ABB RAPID module: c1599a78.mod

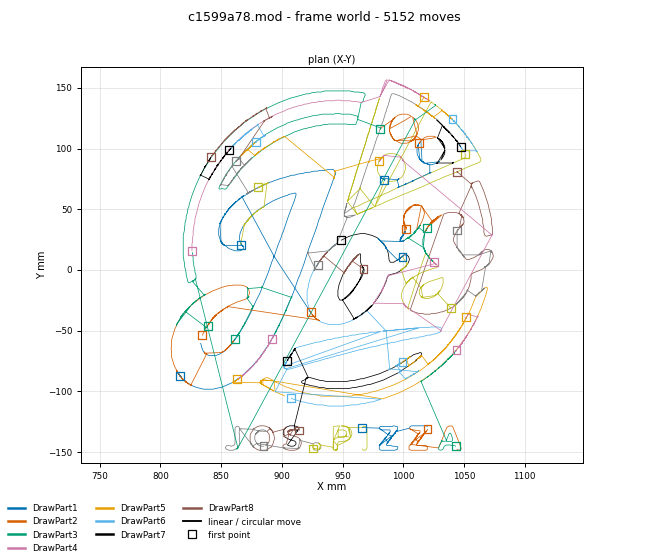
[picture p0: tool path of c1599a78.mod in frame world, 5152 of 5154 moves have a stored position in this frame; points joined in program order, loops and branches not executed]
MODULE ImageDraw
  ! Generated 2026-10-07 06:19 for ABB IRB 1600-10/1.45: 481 strokes
  ! Page 500 x 350 mm. Work object wPaper: Z points up, so pen-up is +Z and the tool uses orientation [0,1,0,0].
  PERS tooldata tPen:=[TRUE,[[0,0,120],[1,0,0,0]],[0.3,[0,0,60],[1,0,0,0],0,0,0]];
  PERS wobjdata wPaper:=[FALSE,TRUE,"",[[700,-175,0],[1,0,0,0]],[[0,0,0],[1,0,0,0]]];
  CONST robtarget pOrigin:=[[0,0,0],[0,1,0,0],[0,0,0,0],[9E9,9E9,9E9,9E9,9E9,9E9]];
  CONST jointtarget jHome:=[[0,0,0,0,30,0],[9E9,9E9,9E9,9E9,9E9,9E9]];
  CONST speeddata vTravel:=[250,200,5000,1000];

  PROC DrawImage()
    SingArea\Wrist;
    ConfL\Off;
    ConfJ\Off;
    MoveAbsJ jHome\NoEOffs,vTravel,fine,tPen;
    DrawPart1;
    DrawPart2;
    DrawPart3;
    DrawPart4;
    DrawPart5;
    DrawPart6;
    DrawPart7;
    DrawPart8;
    DrawPart9;
    DrawPart10;
    DrawPart11;
    DrawPart12;
    DrawPart13;
    DrawPart14;
    DrawPart15;
    DrawPart16;
    DrawPart17;
    DrawPart18;
    DrawPart19;
    DrawPart20;
    DrawPart21;
    DrawPart22;
    DrawPart23;
    DrawPart24;
    DrawPart25;
    DrawPart26;
    DrawPart27;
    DrawPart28;
    DrawPart29;
    DrawPart30;
    DrawPart31;
    DrawPart32;
    DrawPart33;
    DrawPart34;
    DrawPart35;
    DrawPart36;
    DrawPart37;
    DrawPart38;
    DrawPart39;
    DrawPart40;
    DrawPart41;
    DrawPart42;
    DrawPart43;
    MoveAbsJ jHome\NoEOffs,vTravel,fine,tPen;
  ENDPROC

  PROC DrawPart1()
    MoveL Offs(pOrigin,115.92,87.85,6.00),vTravel,z5,tPen\WObj:=wPaper;
    MoveL Offs(pOrigin,115.92,87.85,0.00),v60,z0,tPen\WObj:=wPaper;
    MoveL Offs(pOrigin,116.87,86.89,0.00),v40,z0,tPen\WObj:=wPaper;
    MoveL Offs(pOrigin,116.87,87.37,0.00),v40,z0,tPen\WObj:=wPaper;
    MoveL Offs(pOrigin,116.39,87.37,0.00),v40,z0,tPen\WObj:=wPaper;
    MoveL Offs(pOrigin,115.92,87.85,0.00),v40,z0,tPen\WObj:=wPaper;
    MoveL Offs(pOrigin,116.87,86.89,0.00),v40,z0,tPen\WObj:=wPaper;
    MoveL Offs(pOrigin,116.87,87.37,0.00),v40,z0,tPen\WObj:=wPaper;
    MoveL Offs(pOrigin,116.39,87.37,0.00),v40,z0,tPen\WObj:=wPaper;
    MoveL Offs(pOrigin,115.92,87.85,0.00),v40,z0,tPen\WObj:=wPaper;
    MoveL Offs(pOrigin,115.44,88.80,0.00),v40,z0,tPen\WObj:=wPaper;
    MoveL Offs(pOrigin,115.44,89.28,0.00),v40,z0,tPen\WObj:=wPaper;
    MoveL Offs(pOrigin,114.96,89.28,0.00),v40,z0,tPen\WObj:=wPaper;
    MoveL Offs(pOrigin,114.48,89.76,0.00),v40,z0,tPen\WObj:=wPaper;
    MoveL Offs(pOrigin,115.44,88.80,0.00),v40,z0,tPen\WObj:=wPaper;
    MoveL Offs(pOrigin,115.44,89.28,0.00),v40,z0,tPen\WObj:=wPaper;
    MoveL Offs(pOrigin,114.96,89.28,0.00),v40,z0,tPen\WObj:=wPaper;
    MoveL Offs(pOrigin,114.48,89.76,0.00),v40,z0,tPen\WObj:=wPaper;
    MoveL Offs(pOrigin,115.44,88.80,0.00),v40,fine,tPen\WObj:=wPaper;
    MoveL Offs(pOrigin,115.44,88.80,6.00),v60,z5,tPen\WObj:=wPaper;
    MoveL Offs(pOrigin,114.32,90.72,6.00),vTravel,z5,tPen\WObj:=wPaper;
    MoveL Offs(pOrigin,114.32,90.72,0.00),v60,z0,tPen\WObj:=wPaper;
    MoveL Offs(pOrigin,117.83,85.93,0.00),v40,z0,tPen\WObj:=wPaper;
    MoveL Offs(pOrigin,121.66,82.58,0.00),v40,z0,tPen\WObj:=wPaper;
    MoveL Offs(pOrigin,126.45,79.54,0.00),v40,z0,tPen\WObj:=wPaper;
    MoveL Offs(pOrigin,129.80,78.27,0.00),v40,z0,tPen\WObj:=wPaper;
    MoveL Offs(pOrigin,135.55,76.83,0.00),v40,z0,tPen\WObj:=wPaper;
    MoveL Offs(pOrigin,143.21,76.83,0.00),v40,z0,tPen\WObj:=wPaper;
    MoveL Offs(pOrigin,150.87,78.59,0.00),v40,z0,tPen\WObj:=wPaper;
    MoveL Offs(pOrigin,158.54,81.94,0.00),v40,z0,tPen\WObj:=wPaper;
    MoveL Offs(pOrigin,166.68,87.37,0.00),v40,z0,tPen\WObj:=wPaper;
    MoveL Offs(pOrigin,176.25,96.46,0.00),v40,z0,tPen\WObj:=wPaper;
    MoveL Offs(pOrigin,181.52,102.69,0.00),v40,z0,tPen\WObj:=wPaper;
    MoveL Offs(pOrigin,189.50,114.18,0.00),v40,z0,tPen\WObj:=wPaper;
    MoveL Offs(pOrigin,194.13,122.80,0.00),v40,z0,tPen\WObj:=wPaper;
    MoveL Offs(pOrigin,200.36,135.25,0.00),v40,z0,tPen\WObj:=wPaper;
    MoveL Offs(pOrigin,209.46,156.32,0.00),v40,z0,tPen\WObj:=wPaper;
    MoveL Offs(pOrigin,213.77,168.77,0.00),v40,z0,tPen\WObj:=wPaper;
    MoveL Offs(pOrigin,214.40,169.73,0.00),v40,z0,tPen\WObj:=wPaper;
    MoveL Offs(pOrigin,218.08,179.79,0.00),v40,z0,tPen\WObj:=wPaper;
    MoveL Offs(pOrigin,222.07,192.24,0.00),v40,z0,tPen\WObj:=wPaper;
    MoveL Offs(pOrigin,228.61,209.96,0.00),v40,z0,tPen\WObj:=wPaper;
    MoveL Offs(pOrigin,230.37,216.18,0.00),v40,z0,tPen\WObj:=wPaper;
    MoveL Offs(pOrigin,231.16,217.62,0.00),v40,z0,tPen\WObj:=wPaper;
    MoveL Offs(pOrigin,234.04,226.72,0.00),v40,z0,tPen\WObj:=wPaper;
    MoveL Offs(pOrigin,242.02,248.27,0.00),v40,z0,tPen\WObj:=wPaper;
    MoveL Offs(pOrigin,242.66,250.66,0.00),v40,z0,tPen\WObj:=wPaper;
    MoveL Offs(pOrigin,244.25,254.01,0.00),v40,z0,tPen\WObj:=wPaper;
    MoveL Offs(pOrigin,244.09,255.93,0.00),v40,z0,tPen\WObj:=wPaper;
    MoveL Offs(pOrigin,242.34,257.69,0.00),v40,z0,tPen\WObj:=wPaper;
    MoveL Offs(pOrigin,238.51,257.85,0.00),v40,z0,tPen\WObj:=wPaper;
    MoveL Offs(pOrigin,234.68,256.89,0.00),v40,z0,tPen\WObj:=wPaper;
    MoveL Offs(pOrigin,230.85,256.89,0.00),v40,z0,tPen\WObj:=wPaper;
    MoveL Offs(pOrigin,229.41,256.41,0.00),v40,z0,tPen\WObj:=wPaper;
    MoveL Offs(pOrigin,226.54,256.41,0.00),v40,z0,tPen\WObj:=wPaper;
    MoveL Offs(pOrigin,222.70,255.45,0.00),v40,z0,tPen\WObj:=wPaper;
    MoveL Offs(pOrigin,220.31,255.45,0.00),v40,z0,tPen\WObj:=wPaper;
    MoveL Offs(pOrigin,216.96,254.49,0.00),v40,z0,tPen\WObj:=wPaper;
    MoveL Offs(pOrigin,213.13,254.01,0.00),v40,z0,tPen\WObj:=wPaper;
    MoveL Offs(pOrigin,210.25,253.06,0.00),v40,z0,tPen\WObj:=wPaper;
    MoveL Offs(pOrigin,208.34,253.06,0.00),v40,z0,tPen\WObj:=wPaper;
    MoveL Offs(pOrigin,200.68,250.66,0.00),v40,z0,tPen\WObj:=wPaper;
    MoveL Offs(pOrigin,199.72,250.66,0.00),v40,z0,tPen\WObj:=wPaper;
    MoveL Offs(pOrigin,189.66,246.99,0.00),v40,z0,tPen\WObj:=wPaper;
    MoveL Offs(pOrigin,181.04,242.84,0.00),v40,z0,tPen\WObj:=wPaper;
    MoveL Offs(pOrigin,179.13,242.20,0.00),v40,z0,tPen\WObj:=wPaper;
    MoveL Offs(pOrigin,167.15,234.86,0.00),v40,z0,tPen\WObj:=wPaper;
    MoveL Offs(pOrigin,162.37,231.03,0.00),v40,z0,tPen\WObj:=wPaper;
    MoveL Offs(pOrigin,156.62,225.28,0.00),v40,z0,tPen\WObj:=wPaper;
    MoveL Offs(pOrigin,153.75,221.45,0.00),v40,z0,tPen\WObj:=wPaper;
    MoveL Offs(pOrigin,151.03,217.14,0.00),v40,z0,tPen\WObj:=wPaper;
    MoveL Offs(pOrigin,148.48,210.92,0.00),v40,z0,tPen\WObj:=wPaper;
    MoveL Offs(pOrigin,148.00,208.52,0.00),v40,z0,tPen\WObj:=wPaper;
    MoveL Offs(pOrigin,148.00,203.73,0.00),v40,z0,tPen\WObj:=wPaper;
    MoveL Offs(pOrigin,149.28,199.90,0.00),v40,z0,tPen\WObj:=wPaper;
    MoveL Offs(pOrigin,151.83,196.23,0.00),v40,z0,tPen\WObj:=wPaper;
    MoveL Offs(pOrigin,156.62,192.56,0.00),v40,z0,tPen\WObj:=wPaper;
    MoveL Offs(pOrigin,161.41,190.80,0.00),v40,z0,tPen\WObj:=wPaper;
    MoveL Offs(pOrigin,165.72,190.80,0.00),v40,z0,tPen\WObj:=wPaper;
    MoveL Offs(pOrigin,167.63,191.76,0.00),v40,z0,tPen\WObj:=wPaper;
    MoveL Offs(pOrigin,168.59,193.20,0.00),v40,z0,tPen\WObj:=wPaper;
    MoveL Offs(pOrigin,168.43,194.15,0.00),v40,z0,tPen\WObj:=wPaper;
    MoveL Offs(pOrigin,167.00,195.59,0.00),v40,z0,tPen\WObj:=wPaper;
    MoveL Offs(pOrigin,165.24,199.90,0.00),v40,z0,tPen\WObj:=wPaper;
    MoveL Offs(pOrigin,165.24,203.25,0.00),v40,z0,tPen\WObj:=wPaper;
    MoveL Offs(pOrigin,165.72,205.65,0.00),v40,z0,tPen\WObj:=wPaper;
    MoveL Offs(pOrigin,168.27,211.39,0.00),v40,z0,tPen\WObj:=wPaper;
    MoveL Offs(pOrigin,172.90,217.62,0.00),v40,z0,tPen\WObj:=wPaper;
    MoveL Offs(pOrigin,179.61,223.85,0.00),v40,z0,tPen\WObj:=wPaper;
    MoveL Offs(pOrigin,187.27,228.79,0.00),v40,z0,tPen\WObj:=wPaper;
    MoveL Offs(pOrigin,193.49,232.31,0.00),v40,z0,tPen\WObj:=wPaper;
    MoveL Offs(pOrigin,201.15,235.50,0.00),v40,z0,tPen\WObj:=wPaper;
    MoveL Offs(pOrigin,204.51,236.46,0.00),v40,z0,tPen\WObj:=wPaper;
    MoveL Offs(pOrigin,205.94,237.25,0.00),v40,z0,tPen\WObj:=wPaper;
    MoveL Offs(pOrigin,210.73,238.37,0.00),v40,z0,tPen\WObj:=wPaper;
    MoveL Offs(pOrigin,211.53,238.21,0.00),v40,z0,tPen\WObj:=wPaper;
    MoveL Offs(pOrigin,211.69,236.77,0.00),v40,z0,tPen\WObj:=wPaper;
    MoveL Offs(pOrigin,210.41,232.46,0.00),v40,z0,tPen\WObj:=wPaper;
    MoveL Offs(pOrigin,205.31,219.06,0.00),v40,z0,tPen\WObj:=wPaper;
    MoveL Offs(pOrigin,201.00,206.13,0.00),v40,z0,tPen\WObj:=wPaper;
    MoveL Offs(pOrigin,200.36,205.17,0.00),v40,z0,tPen\WObj:=wPaper;
    MoveL Offs(pOrigin,199.40,201.82,0.00),v40,z0,tPen\WObj:=wPaper;
    MoveL Offs(pOrigin,196.69,195.11,0.00),v40,z0,tPen\WObj:=wPaper;
    MoveL Offs(pOrigin,193.65,186.01,0.00),v40,z0,tPen\WObj:=wPaper;
    MoveL Offs(pOrigin,191.74,181.70,0.00),v40,z0,tPen\WObj:=wPaper;
    MoveL Offs(pOrigin,188.86,173.08,0.00),v40,z0,tPen\WObj:=wPaper;
    MoveL Offs(pOrigin,181.68,155.37,0.00),v40,z0,tPen\WObj:=wPaper;
    MoveL Offs(pOrigin,178.49,149.14,0.00),v40,z0,tPen\WObj:=wPaper;
    MoveL Offs(pOrigin,174.50,140.04,0.00),v40,z0,tPen\WObj:=wPaper;
    MoveL Offs(pOrigin,169.23,129.99,0.00),v40,z0,tPen\WObj:=wPaper;
    MoveL Offs(pOrigin,163.48,120.41,0.00),v40,z0,tPen\WObj:=wPaper;
    MoveL Offs(pOrigin,158.54,113.70,0.00),v40,z0,tPen\WObj:=wPaper;
    MoveL Offs(pOrigin,153.27,108.44,0.00),v40,z0,tPen\WObj:=wPaper;
    MoveL Offs(pOrigin,148.00,105.40,0.00),v40,z0,tPen\WObj:=wPaper;
    MoveL Offs(pOrigin,145.61,104.61,0.00),v40,z0,tPen\WObj:=wPaper;
    MoveL Offs(pOrigin,139.86,104.61,0.00),v40,z0,tPen\WObj:=wPaper;
    MoveL Offs(pOrigin,137.46,105.72,0.00),v40,z0,tPen\WObj:=wPaper;
    MoveL Offs(pOrigin,135.71,107.48,0.00),v40,z0,tPen\WObj:=wPaper;
    MoveL Offs(pOrigin,134.59,109.39,0.00),v40,z0,tPen\WObj:=wPaper;
    MoveL Offs(pOrigin,133.15,114.66,0.00),v40,z0,tPen\WObj:=wPaper;
  ENDPROC

  PROC DrawPart2()
    MoveL Offs(pOrigin,134.59,121.37,0.00),v40,z0,tPen\WObj:=wPaper;
    MoveL Offs(pOrigin,137.15,127.11,0.00),v40,z0,tPen\WObj:=wPaper;
    MoveL Offs(pOrigin,143.21,135.73,0.00),v40,z0,tPen\WObj:=wPaper;
    MoveL Offs(pOrigin,145.61,138.13,0.00),v40,z0,tPen\WObj:=wPaper;
    MoveL Offs(pOrigin,149.92,141.48,0.00),v40,z0,tPen\WObj:=wPaper;
    MoveL Offs(pOrigin,155.66,145.15,0.00),v40,z0,tPen\WObj:=wPaper;
    MoveL Offs(pOrigin,162.85,148.50,0.00),v40,z0,tPen\WObj:=wPaper;
    MoveL Offs(pOrigin,170.03,150.90,0.00),v40,z0,tPen\WObj:=wPaper;
    MoveL Offs(pOrigin,172.42,152.97,0.00),v40,z0,tPen\WObj:=wPaper;
    MoveL Offs(pOrigin,173.38,156.32,0.00),v40,z0,tPen\WObj:=wPaper;
    MoveL Offs(pOrigin,172.58,159.20,0.00),v40,z0,tPen\WObj:=wPaper;
    MoveL Offs(pOrigin,170.51,161.43,0.00),v40,z0,tPen\WObj:=wPaper;
    MoveL Offs(pOrigin,166.68,162.55,0.00),v40,z0,tPen\WObj:=wPaper;
    MoveL Offs(pOrigin,159.97,162.55,0.00),v40,z0,tPen\WObj:=wPaper;
    MoveL Offs(pOrigin,158.54,162.07,0.00),v40,z0,tPen\WObj:=wPaper;
    MoveL Offs(pOrigin,155.66,162.07,0.00),v40,z0,tPen\WObj:=wPaper;
    MoveL Offs(pOrigin,150.87,160.79,0.00),v40,z0,tPen\WObj:=wPaper;
    MoveL Offs(pOrigin,142.25,157.44,0.00),v40,z0,tPen\WObj:=wPaper;
    MoveL Offs(pOrigin,135.07,153.45,0.00),v40,z0,tPen\WObj:=wPaper;
    MoveL Offs(pOrigin,125.01,145.79,0.00),v40,z0,tPen\WObj:=wPaper;
    MoveL Offs(pOrigin,124.06,144.35,0.00),v40,z0,tPen\WObj:=wPaper;
    MoveL Offs(pOrigin,118.79,138.61,0.00),v40,z0,tPen\WObj:=wPaper;
    MoveL Offs(pOrigin,115.28,133.34,0.00),v40,z0,tPen\WObj:=wPaper;
    MoveL Offs(pOrigin,111.77,126.15,0.00),v40,z0,tPen\WObj:=wPaper;
    MoveL Offs(pOrigin,109.21,117.54,0.00),v40,z0,tPen\WObj:=wPaper;
    MoveL Offs(pOrigin,109.21,111.79,0.00),v40,z0,tPen\WObj:=wPaper;
    MoveL Offs(pOrigin,108.73,110.35,0.00),v40,z0,tPen\WObj:=wPaper;
    MoveL Offs(pOrigin,109.21,108.44,0.00),v40,z0,tPen\WObj:=wPaper;
    MoveL Offs(pOrigin,109.21,103.17,0.00),v40,z0,tPen\WObj:=wPaper;
    MoveL Offs(pOrigin,111.45,95.99,0.00),v40,z0,tPen\WObj:=wPaper;
    MoveL Offs(pOrigin,114.32,90.72,0.00),v40,fine,tPen\WObj:=wPaper;
    MoveL Offs(pOrigin,114.32,90.72,6.00),v60,z5,tPen\WObj:=wPaper;
    MoveL Offs(pOrigin,113.52,91.68,6.00),vTravel,z5,tPen\WObj:=wPaper;
    MoveL Offs(pOrigin,113.52,91.68,0.00),v60,z0,tPen\WObj:=wPaper;
    MoveL Offs(pOrigin,113.52,92.15,0.00),v40,z0,tPen\WObj:=wPaper;
    MoveL Offs(pOrigin,113.04,92.15,0.00),v40,z0,tPen\WObj:=wPaper;
    MoveL Offs(pOrigin,113.52,91.68,0.00),v40,z0,tPen\WObj:=wPaper;
    MoveL Offs(pOrigin,113.52,92.15,0.00),v40,z0,tPen\WObj:=wPaper;
    MoveL Offs(pOrigin,113.04,92.15,0.00),v40,z0,tPen\WObj:=wPaper;
    MoveL Offs(pOrigin,113.52,91.68,0.00),v40,fine,tPen\WObj:=wPaper;
    MoveL Offs(pOrigin,113.52,91.68,6.00),v60,z5,tPen\WObj:=wPaper;
    MoveL Offs(pOrigin,117.35,85.93,6.00),vTravel,z5,tPen\WObj:=wPaper;
    MoveL Offs(pOrigin,117.35,85.93,0.00),v60,z0,tPen\WObj:=wPaper;
    MoveL Offs(pOrigin,119.27,84.01,0.00),v40,z0,tPen\WObj:=wPaper;
    MoveL Offs(pOrigin,119.27,84.49,0.00),v40,z0,tPen\WObj:=wPaper;
    MoveL Offs(pOrigin,118.79,84.49,0.00),v40,z0,tPen\WObj:=wPaper;
    MoveL Offs(pOrigin,117.35,85.93,0.00),v40,z0,tPen\WObj:=wPaper;
    MoveL Offs(pOrigin,119.27,84.01,0.00),v40,z0,tPen\WObj:=wPaper;
    MoveL Offs(pOrigin,119.27,84.49,0.00),v40,z0,tPen\WObj:=wPaper;
    MoveL Offs(pOrigin,118.79,84.49,0.00),v40,z0,tPen\WObj:=wPaper;
    MoveL Offs(pOrigin,117.35,85.93,0.00),v40,fine,tPen\WObj:=wPaper;
    MoveL Offs(pOrigin,117.35,85.93,6.00),v60,z5,tPen\WObj:=wPaper;
    MoveL Offs(pOrigin,120.23,83.54,6.00),vTravel,z5,tPen\WObj:=wPaper;
    MoveL Offs(pOrigin,120.23,83.54,0.00),v60,z0,tPen\WObj:=wPaper;
    MoveL Offs(pOrigin,121.66,82.10,0.00),v40,z0,tPen\WObj:=wPaper;
    MoveL Offs(pOrigin,121.66,82.58,0.00),v40,z0,tPen\WObj:=wPaper;
    MoveL Offs(pOrigin,121.18,82.58,0.00),v40,z0,tPen\WObj:=wPaper;
    MoveL Offs(pOrigin,120.23,83.54,0.00),v40,z0,tPen\WObj:=wPaper;
    MoveL Offs(pOrigin,121.66,82.10,0.00),v40,z0,tPen\WObj:=wPaper;
    MoveL Offs(pOrigin,121.66,82.58,0.00),v40,z0,tPen\WObj:=wPaper;
    MoveL Offs(pOrigin,121.18,82.58,0.00),v40,z0,tPen\WObj:=wPaper;
    MoveL Offs(pOrigin,120.23,83.54,0.00),v40,fine,tPen\WObj:=wPaper;
    MoveL Offs(pOrigin,120.23,83.54,6.00),v60,z5,tPen\WObj:=wPaper;
    MoveL Offs(pOrigin,122.62,81.62,6.00),vTravel,z5,tPen\WObj:=wPaper;
    MoveL Offs(pOrigin,122.62,81.62,0.00),v60,z0,tPen\WObj:=wPaper;
    MoveL Offs(pOrigin,123.10,81.14,0.00),v40,z0,tPen\WObj:=wPaper;
    MoveL Offs(pOrigin,123.10,81.62,0.00),v40,z0,tPen\WObj:=wPaper;
    MoveL Offs(pOrigin,122.62,81.62,0.00),v40,z0,tPen\WObj:=wPaper;
    MoveL Offs(pOrigin,123.10,81.14,0.00),v40,z0,tPen\WObj:=wPaper;
    MoveL Offs(pOrigin,123.10,81.62,0.00),v40,z0,tPen\WObj:=wPaper;
    MoveL Offs(pOrigin,122.62,81.62,0.00),v40,fine,tPen\WObj:=wPaper;
    MoveL Offs(pOrigin,122.62,81.62,6.00),v60,z5,tPen\WObj:=wPaper;
    MoveL Offs(pOrigin,125.01,80.18,6.00),vTravel,z5,tPen\WObj:=wPaper;
    MoveL Offs(pOrigin,125.01,80.18,0.00),v60,z0,tPen\WObj:=wPaper;
    MoveL Offs(pOrigin,125.49,79.70,0.00),v40,z0,tPen\WObj:=wPaper;
    MoveL Offs(pOrigin,125.49,80.18,0.00),v40,z0,tPen\WObj:=wPaper;
    MoveL Offs(pOrigin,125.01,80.18,0.00),v40,z0,tPen\WObj:=wPaper;
    MoveL Offs(pOrigin,125.49,79.70,0.00),v40,z0,tPen\WObj:=wPaper;
    MoveL Offs(pOrigin,125.49,80.18,0.00),v40,z0,tPen\WObj:=wPaper;
    MoveL Offs(pOrigin,125.01,80.18,0.00),v40,fine,tPen\WObj:=wPaper;
    MoveL Offs(pOrigin,125.01,80.18,6.00),v60,z5,tPen\WObj:=wPaper;
    MoveL Offs(pOrigin,137.94,105.56,6.00),vTravel,z5,tPen\WObj:=wPaper;
    MoveL Offs(pOrigin,137.94,105.56,0.00),v60,z0,tPen\WObj:=wPaper;
    MoveL Offs(pOrigin,138.42,105.56,0.00),v40,z0,tPen\WObj:=wPaper;
    MoveL Offs(pOrigin,137.46,106.04,0.00),v40,z0,tPen\WObj:=wPaper;
    MoveL Offs(pOrigin,137.94,105.56,0.00),v40,z0,tPen\WObj:=wPaper;
    MoveL Offs(pOrigin,138.42,105.56,0.00),v40,z0,tPen\WObj:=wPaper;
    MoveL Offs(pOrigin,137.46,106.04,0.00),v40,z0,tPen\WObj:=wPaper;
    MoveL Offs(pOrigin,137.94,105.56,0.00),v40,fine,tPen\WObj:=wPaper;
    MoveL Offs(pOrigin,137.94,105.56,6.00),v60,z5,tPen\WObj:=wPaper;
    MoveL Offs(pOrigin,136.51,106.52,6.00),vTravel,z5,tPen\WObj:=wPaper;
    MoveL Offs(pOrigin,136.51,106.52,0.00),v60,z0,tPen\WObj:=wPaper;
    MoveL Offs(pOrigin,136.03,107.48,0.00),v40,z0,tPen\WObj:=wPaper;
    MoveL Offs(pOrigin,136.51,107.00,0.00),v40,z0,tPen\WObj:=wPaper;
    MoveL Offs(pOrigin,136.51,106.52,0.00),v40,z0,tPen\WObj:=wPaper;
    MoveL Offs(pOrigin,136.03,107.48,0.00),v40,z0,tPen\WObj:=wPaper;
    MoveL Offs(pOrigin,136.51,107.00,0.00),v40,z0,tPen\WObj:=wPaper;
    MoveL Offs(pOrigin,136.51,106.52,0.00),v40,fine,tPen\WObj:=wPaper;
    MoveL Offs(pOrigin,136.51,106.52,6.00),v60,z5,tPen\WObj:=wPaper;
    MoveL Offs(pOrigin,150.39,107.00,6.00),vTravel,z5,tPen\WObj:=wPaper;
    MoveL Offs(pOrigin,150.39,107.00,0.00),v60,z0,tPen\WObj:=wPaper;
    MoveL Offs(pOrigin,150.87,107.00,0.00),v40,z0,tPen\WObj:=wPaper;
    MoveL Offs(pOrigin,151.83,107.96,0.00),v40,z0,tPen\WObj:=wPaper;
    MoveL Offs(pOrigin,150.39,107.00,0.00),v40,z0,tPen\WObj:=wPaper;
    MoveL Offs(pOrigin,150.87,107.00,0.00),v40,z0,tPen\WObj:=wPaper;
    MoveL Offs(pOrigin,151.83,107.96,0.00),v40,z0,tPen\WObj:=wPaper;
    MoveL Offs(pOrigin,150.39,107.00,0.00),v40,fine,tPen\WObj:=wPaper;
    MoveL Offs(pOrigin,150.39,107.00,6.00),v60,z5,tPen\WObj:=wPaper;
    MoveL Offs(pOrigin,153.27,108.92,6.00),vTravel,z5,tPen\WObj:=wPaper;
    MoveL Offs(pOrigin,153.27,108.92,0.00),v60,z0,tPen\WObj:=wPaper;
    MoveL Offs(pOrigin,157.58,113.23,0.00),v40,z0,tPen\WObj:=wPaper;
    MoveL Offs(pOrigin,153.27,108.92,0.00),v40,fine,tPen\WObj:=wPaper;
    MoveL Offs(pOrigin,153.27,108.92,6.00),v60,z5,tPen\WObj:=wPaper;
    MoveL Offs(pOrigin,158.54,114.18,6.00),vTravel,z5,tPen\WObj:=wPaper;
    MoveL Offs(pOrigin,158.54,114.18,0.00),v60,z0,tPen\WObj:=wPaper;
    MoveL Offs(pOrigin,159.97,116.10,0.00),v40,z0,tPen\WObj:=wPaper;
    MoveL Offs(pOrigin,158.54,114.18,0.00),v40,fine,tPen\WObj:=wPaper;
    MoveL Offs(pOrigin,158.54,114.18,6.00),v60,z5,tPen\WObj:=wPaper;
    MoveL Offs(pOrigin,160.45,117.06,6.00),vTravel,z5,tPen\WObj:=wPaper;
    MoveL Offs(pOrigin,160.45,117.06,0.00),v60,z0,tPen\WObj:=wPaper;
  ENDPROC

  PROC DrawPart3()
    MoveL Offs(pOrigin,161.41,118.01,0.00),v40,z0,tPen\WObj:=wPaper;
    MoveL Offs(pOrigin,160.45,117.06,0.00),v40,fine,tPen\WObj:=wPaper;
    MoveL Offs(pOrigin,160.45,117.06,6.00),v60,z5,tPen\WObj:=wPaper;
    MoveL Offs(pOrigin,163.32,120.89,6.00),vTravel,z5,tPen\WObj:=wPaper;
    MoveL Offs(pOrigin,163.32,120.89,0.00),v60,z0,tPen\WObj:=wPaper;
    MoveL Offs(pOrigin,163.80,121.37,0.00),v40,z0,tPen\WObj:=wPaper;
    MoveL Offs(pOrigin,163.80,121.85,0.00),v40,z0,tPen\WObj:=wPaper;
    MoveL Offs(pOrigin,163.32,120.89,0.00),v40,z0,tPen\WObj:=wPaper;
    MoveL Offs(pOrigin,163.80,121.37,0.00),v40,z0,tPen\WObj:=wPaper;
    MoveL Offs(pOrigin,163.80,121.85,0.00),v40,z0,tPen\WObj:=wPaper;
    MoveL Offs(pOrigin,163.32,120.89,0.00),v40,fine,tPen\WObj:=wPaper;
    MoveL Offs(pOrigin,163.32,120.89,6.00),v60,z5,tPen\WObj:=wPaper;
    MoveL Offs(pOrigin,164.28,122.32,6.00),vTravel,z5,tPen\WObj:=wPaper;
    MoveL Offs(pOrigin,164.28,122.32,0.00),v60,z0,tPen\WObj:=wPaper;
    MoveL Offs(pOrigin,164.76,122.80,0.00),v40,z0,tPen\WObj:=wPaper;
    MoveL Offs(pOrigin,164.76,123.28,0.00),v40,z0,tPen\WObj:=wPaper;
    MoveL Offs(pOrigin,164.28,122.32,0.00),v40,z0,tPen\WObj:=wPaper;
    MoveL Offs(pOrigin,164.76,122.80,0.00),v40,z0,tPen\WObj:=wPaper;
    MoveL Offs(pOrigin,164.76,123.28,0.00),v40,z0,tPen\WObj:=wPaper;
    MoveL Offs(pOrigin,164.28,122.32,0.00),v40,fine,tPen\WObj:=wPaper;
    MoveL Offs(pOrigin,164.28,122.32,6.00),v60,z5,tPen\WObj:=wPaper;
    MoveL Offs(pOrigin,167.63,128.07,6.00),vTravel,z5,tPen\WObj:=wPaper;
    MoveL Offs(pOrigin,167.63,128.07,0.00),v60,z0,tPen\WObj:=wPaper;
    MoveL Offs(pOrigin,168.59,129.51,0.00),v40,z0,tPen\WObj:=wPaper;
    MoveL Offs(pOrigin,167.63,128.07,0.00),v40,fine,tPen\WObj:=wPaper;
    MoveL Offs(pOrigin,167.63,128.07,6.00),v60,z5,tPen\WObj:=wPaper;
    MoveL Offs(pOrigin,169.07,130.46,6.00),vTravel,z5,tPen\WObj:=wPaper;
    MoveL Offs(pOrigin,169.07,130.46,0.00),v60,z0,tPen\WObj:=wPaper;
    MoveL Offs(pOrigin,169.55,130.94,0.00),v40,z0,tPen\WObj:=wPaper;
    MoveL Offs(pOrigin,169.55,131.42,0.00),v40,z0,tPen\WObj:=wPaper;
    MoveL Offs(pOrigin,169.07,130.46,0.00),v40,z0,tPen\WObj:=wPaper;
    MoveL Offs(pOrigin,169.55,130.94,0.00),v40,z0,tPen\WObj:=wPaper;
    MoveL Offs(pOrigin,169.55,131.42,0.00),v40,z0,tPen\WObj:=wPaper;
    MoveL Offs(pOrigin,169.07,130.46,0.00),v40,fine,tPen\WObj:=wPaper;
    MoveL Offs(pOrigin,169.07,130.46,6.00),v60,z5,tPen\WObj:=wPaper;
    MoveL Offs(pOrigin,175.30,142.92,6.00),vTravel,z5,tPen\WObj:=wPaper;
    MoveL Offs(pOrigin,175.30,142.92,0.00),v60,z0,tPen\WObj:=wPaper;
    MoveL Offs(pOrigin,175.77,143.39,0.00),v40,z0,tPen\WObj:=wPaper;
    MoveL Offs(pOrigin,175.77,143.87,0.00),v40,z0,tPen\WObj:=wPaper;
    MoveL Offs(pOrigin,175.30,142.92,0.00),v40,z0,tPen\WObj:=wPaper;
    MoveL Offs(pOrigin,175.77,143.39,0.00),v40,z0,tPen\WObj:=wPaper;
    MoveL Offs(pOrigin,175.77,143.87,0.00),v40,z0,tPen\WObj:=wPaper;
    MoveL Offs(pOrigin,175.30,142.92,0.00),v40,fine,tPen\WObj:=wPaper;
    MoveL Offs(pOrigin,175.30,142.92,6.00),v60,z5,tPen\WObj:=wPaper;
    MoveL Offs(pOrigin,176.25,144.83,6.00),vTravel,z5,tPen\WObj:=wPaper;
    MoveL Offs(pOrigin,176.25,144.83,0.00),v60,z0,tPen\WObj:=wPaper;
    MoveL Offs(pOrigin,176.73,145.31,0.00),v40,z0,tPen\WObj:=wPaper;
    MoveL Offs(pOrigin,176.73,145.79,0.00),v40,z0,tPen\WObj:=wPaper;
    MoveL Offs(pOrigin,176.25,144.83,0.00),v40,z0,tPen\WObj:=wPaper;
    MoveL Offs(pOrigin,176.73,145.31,0.00),v40,z0,tPen\WObj:=wPaper;
    MoveL Offs(pOrigin,176.73,145.79,0.00),v40,z0,tPen\WObj:=wPaper;
    MoveL Offs(pOrigin,176.25,144.83,0.00),v40,fine,tPen\WObj:=wPaper;
    MoveL Offs(pOrigin,176.25,144.83,6.00),v60,z5,tPen\WObj:=wPaper;
    MoveL Offs(pOrigin,171.46,151.54,6.00),vTravel,z5,tPen\WObj:=wPaper;
    MoveL Offs(pOrigin,171.46,151.54,0.00),v60,z0,tPen\WObj:=wPaper;
    MoveL Offs(pOrigin,171.46,152.01,0.00),v40,z0,tPen\WObj:=wPaper;
    MoveL Offs(pOrigin,171.94,152.01,0.00),v40,z0,tPen\WObj:=wPaper;
    MoveL Offs(pOrigin,172.90,152.97,0.00),v40,z0,tPen\WObj:=wPaper;
    MoveL Offs(pOrigin,171.46,151.54,0.00),v40,z0,tPen\WObj:=wPaper;
    MoveL Offs(pOrigin,171.46,152.01,0.00),v40,z0,tPen\WObj:=wPaper;
    MoveL Offs(pOrigin,171.94,152.01,0.00),v40,z0,tPen\WObj:=wPaper;
    MoveL Offs(pOrigin,172.90,152.97,0.00),v40,z0,tPen\WObj:=wPaper;
    MoveL Offs(pOrigin,171.46,151.54,0.00),v40,fine,tPen\WObj:=wPaper;
    MoveL Offs(pOrigin,171.46,151.54,6.00),v60,z5,tPen\WObj:=wPaper;
    MoveL Offs(pOrigin,171.94,159.68,6.00),vTravel,z5,tPen\WObj:=wPaper;
    MoveL Offs(pOrigin,171.94,159.68,0.00),v60,z0,tPen\WObj:=wPaper;
    MoveL Offs(pOrigin,171.46,160.63,0.00),v40,z0,tPen\WObj:=wPaper;
    MoveL Offs(pOrigin,171.94,160.15,0.00),v40,z0,tPen\WObj:=wPaper;
    MoveL Offs(pOrigin,171.94,159.68,0.00),v40,z0,tPen\WObj:=wPaper;
    MoveL Offs(pOrigin,171.46,160.63,0.00),v40,z0,tPen\WObj:=wPaper;
    MoveL Offs(pOrigin,171.94,160.15,0.00),v40,z0,tPen\WObj:=wPaper;
    MoveL Offs(pOrigin,171.94,159.68,0.00),v40,fine,tPen\WObj:=wPaper;
    MoveL Offs(pOrigin,171.94,159.68,6.00),v60,z5,tPen\WObj:=wPaper;
    MoveL Offs(pOrigin,183.44,160.63,6.00),vTravel,z5,tPen\WObj:=wPaper;
    MoveL Offs(pOrigin,183.44,160.63,0.00),v60,z0,tPen\WObj:=wPaper;
    MoveL Offs(pOrigin,183.92,161.11,0.00),v40,z0,tPen\WObj:=wPaper;
    MoveL Offs(pOrigin,183.92,161.59,0.00),v40,z0,tPen\WObj:=wPaper;
    MoveL Offs(pOrigin,183.44,160.63,0.00),v40,z0,tPen\WObj:=wPaper;
    MoveL Offs(pOrigin,183.92,161.11,0.00),v40,z0,tPen\WObj:=wPaper;
    MoveL Offs(pOrigin,183.92,161.59,0.00),v40,z0,tPen\WObj:=wPaper;
    MoveL Offs(pOrigin,183.44,160.63,0.00),v40,fine,tPen\WObj:=wPaper;
    MoveL Offs(pOrigin,183.44,160.63,6.00),v60,z5,tPen\WObj:=wPaper;
    MoveL Offs(pOrigin,207.86,152.49,6.00),vTravel,z5,tPen\WObj:=wPaper;
    MoveL Offs(pOrigin,207.86,152.49,0.00),v60,z0,tPen\WObj:=wPaper;
    MoveL Offs(pOrigin,208.34,152.97,0.00),v40,z0,tPen\WObj:=wPaper;
    MoveL Offs(pOrigin,207.86,152.01,0.00),v40,z0,tPen\WObj:=wPaper;
    MoveL Offs(pOrigin,207.86,152.49,0.00),v40,z0,tPen\WObj:=wPaper;
    MoveL Offs(pOrigin,208.34,152.97,0.00),v40,z0,tPen\WObj:=wPaper;
    MoveL Offs(pOrigin,207.86,152.01,0.00),v40,z0,tPen\WObj:=wPaper;
    MoveL Offs(pOrigin,207.86,152.49,0.00),v40,fine,tPen\WObj:=wPaper;
    MoveL Offs(pOrigin,207.86,152.49,6.00),v60,z5,tPen\WObj:=wPaper;
    MoveL Offs(pOrigin,203.55,141.96,6.00),vTravel,z5,tPen\WObj:=wPaper;
    MoveL Offs(pOrigin,203.55,141.96,0.00),v60,z0,tPen\WObj:=wPaper;
    MoveL Offs(pOrigin,203.07,141.00,0.00),v40,z0,tPen\WObj:=wPaper;
    MoveL Offs(pOrigin,203.07,141.48,0.00),v40,z0,tPen\WObj:=wPaper;
    MoveL Offs(pOrigin,203.55,141.96,0.00),v40,z0,tPen\WObj:=wPaper;
    MoveL Offs(pOrigin,203.07,141.00,0.00),v40,z0,tPen\WObj:=wPaper;
    MoveL Offs(pOrigin,203.07,141.48,0.00),v40,z0,tPen\WObj:=wPaper;
    MoveL Offs(pOrigin,203.55,141.96,0.00),v40,fine,tPen\WObj:=wPaper;
    MoveL Offs(pOrigin,203.55,141.96,6.00),v60,z5,tPen\WObj:=wPaper;
    MoveL Offs(pOrigin,197.80,129.51,6.00),vTravel,z5,tPen\WObj:=wPaper;
    MoveL Offs(pOrigin,197.80,129.51,0.00),v60,z0,tPen\WObj:=wPaper;
    MoveL Offs(pOrigin,197.32,128.55,0.00),v40,z0,tPen\WObj:=wPaper;
    MoveL Offs(pOrigin,197.32,129.03,0.00),v40,z0,tPen\WObj:=wPaper;
    MoveL Offs(pOrigin,197.80,129.51,0.00),v40,z0,tPen\WObj:=wPaper;
    MoveL Offs(pOrigin,197.32,128.55,0.00),v40,z0,tPen\WObj:=wPaper;
    MoveL Offs(pOrigin,197.32,129.03,0.00),v40,z0,tPen\WObj:=wPaper;
    MoveL Offs(pOrigin,197.80,129.51,0.00),v40,fine,tPen\WObj:=wPaper;
    MoveL Offs(pOrigin,197.80,129.51,6.00),v60,z5,tPen\WObj:=wPaper;
    MoveL Offs(pOrigin,195.41,124.72,6.00),vTravel,z5,tPen\WObj:=wPaper;
    MoveL Offs(pOrigin,195.41,124.72,0.00),v60,z0,tPen\WObj:=wPaper;
    MoveL Offs(pOrigin,194.93,123.76,0.00),v40,z0,tPen\WObj:=wPaper;
    MoveL Offs(pOrigin,194.93,124.24,0.00),v40,z0,tPen\WObj:=wPaper;
    MoveL Offs(pOrigin,195.41,124.72,0.00),v40,z0,tPen\WObj:=wPaper;
    MoveL Offs(pOrigin,194.93,123.76,0.00),v40,z0,tPen\WObj:=wPaper;
    MoveL Offs(pOrigin,194.93,124.24,0.00),v40,z0,tPen\WObj:=wPaper;
    MoveL Offs(pOrigin,195.41,124.72,0.00),v40,fine,tPen\WObj:=wPaper;
    MoveL Offs(pOrigin,195.41,124.72,6.00),v60,z5,tPen\WObj:=wPaper;
    MoveL Offs(pOrigin,193.01,119.93,6.00),vTravel,z5,tPen\WObj:=wPaper;
    MoveL Offs(pOrigin,193.01,119.93,0.00),v60,z0,tPen\WObj:=wPaper;
  ENDPROC

  PROC DrawPart4()
    MoveL Offs(pOrigin,192.06,118.49,0.00),v40,z0,tPen\WObj:=wPaper;
    MoveL Offs(pOrigin,192.06,118.97,0.00),v40,z0,tPen\WObj:=wPaper;
    MoveL Offs(pOrigin,193.01,119.93,0.00),v40,z0,tPen\WObj:=wPaper;
    MoveL Offs(pOrigin,192.06,118.49,0.00),v40,z0,tPen\WObj:=wPaper;
    MoveL Offs(pOrigin,192.06,118.97,0.00),v40,z0,tPen\WObj:=wPaper;
    MoveL Offs(pOrigin,193.01,119.93,0.00),v40,fine,tPen\WObj:=wPaper;
    MoveL Offs(pOrigin,193.01,119.93,6.00),v60,z5,tPen\WObj:=wPaper;
    MoveL Offs(pOrigin,191.58,117.54,6.00),vTravel,z5,tPen\WObj:=wPaper;
    MoveL Offs(pOrigin,191.58,117.54,0.00),v60,z0,tPen\WObj:=wPaper;
    MoveL Offs(pOrigin,191.10,116.58,0.00),v40,z0,tPen\WObj:=wPaper;
    MoveL Offs(pOrigin,191.10,117.06,0.00),v40,z0,tPen\WObj:=wPaper;
    MoveL Offs(pOrigin,191.58,117.54,0.00),v40,z0,tPen\WObj:=wPaper;
    MoveL Offs(pOrigin,191.10,116.58,0.00),v40,z0,tPen\WObj:=wPaper;
    MoveL Offs(pOrigin,191.10,117.06,0.00),v40,z0,tPen\WObj:=wPaper;
    MoveL Offs(pOrigin,191.58,117.54,0.00),v40,fine,tPen\WObj:=wPaper;
    MoveL Offs(pOrigin,191.58,117.54,6.00),v60,z5,tPen\WObj:=wPaper;
    MoveL Offs(pOrigin,189.18,113.23,6.00),vTravel,z5,tPen\WObj:=wPaper;
    MoveL Offs(pOrigin,189.18,113.23,0.00),v60,z0,tPen\WObj:=wPaper;
    MoveL Offs(pOrigin,188.23,111.79,0.00),v40,z0,tPen\WObj:=wPaper;
    MoveL Offs(pOrigin,188.23,112.27,0.00),v40,z0,tPen\WObj:=wPaper;
    MoveL Offs(pOrigin,189.18,113.23,0.00),v40,z0,tPen\WObj:=wPaper;
    MoveL Offs(pOrigin,188.23,111.79,0.00),v40,z0,tPen\WObj:=wPaper;
    MoveL Offs(pOrigin,188.23,112.27,0.00),v40,z0,tPen\WObj:=wPaper;
    MoveL Offs(pOrigin,189.18,113.23,0.00),v40,fine,tPen\WObj:=wPaper;
    MoveL Offs(pOrigin,189.18,113.23,6.00),v60,z5,tPen\WObj:=wPaper;
    MoveL Offs(pOrigin,186.31,108.92,6.00),vTravel,z5,tPen\WObj:=wPaper;
    MoveL Offs(pOrigin,186.31,108.92,0.00),v60,z0,tPen\WObj:=wPaper;
    MoveL Offs(pOrigin,185.83,108.44,0.00),v40,z0,tPen\WObj:=wPaper;
    MoveL Offs(pOrigin,185.83,108.92,0.00),v40,z0,tPen\WObj:=wPaper;
    MoveL Offs(pOrigin,186.31,108.92,0.00),v40,z0,tPen\WObj:=wPaper;
    MoveL Offs(pOrigin,185.83,108.44,0.00),v40,z0,tPen\WObj:=wPaper;
    MoveL Offs(pOrigin,185.83,108.92,0.00),v40,z0,tPen\WObj:=wPaper;
    MoveL Offs(pOrigin,186.31,108.92,0.00),v40,fine,tPen\WObj:=wPaper;
    MoveL Offs(pOrigin,186.31,108.92,6.00),v60,z5,tPen\WObj:=wPaper;
    MoveL Offs(pOrigin,185.35,107.48,6.00),vTravel,z5,tPen\WObj:=wPaper;
    MoveL Offs(pOrigin,185.35,107.48,0.00),v60,z0,tPen\WObj:=wPaper;
    MoveL Offs(pOrigin,184.87,107.00,0.00),v40,z0,tPen\WObj:=wPaper;
    MoveL Offs(pOrigin,184.87,107.48,0.00),v40,z0,tPen\WObj:=wPaper;
    MoveL Offs(pOrigin,185.35,107.48,0.00),v40,z0,tPen\WObj:=wPaper;
    MoveL Offs(pOrigin,184.87,107.00,0.00),v40,z0,tPen\WObj:=wPaper;
    MoveL Offs(pOrigin,184.87,107.48,0.00),v40,z0,tPen\WObj:=wPaper;
    MoveL Offs(pOrigin,185.35,107.48,0.00),v40,fine,tPen\WObj:=wPaper;
    MoveL Offs(pOrigin,185.35,107.48,6.00),v60,z5,tPen\WObj:=wPaper;
    MoveL Offs(pOrigin,184.39,106.04,6.00),vTravel,z5,tPen\WObj:=wPaper;
    MoveL Offs(pOrigin,184.39,106.04,0.00),v60,z0,tPen\WObj:=wPaper;
    MoveL Offs(pOrigin,183.92,105.56,0.00),v40,z0,tPen\WObj:=wPaper;
    MoveL Offs(pOrigin,183.92,106.04,0.00),v40,z0,tPen\WObj:=wPaper;
    MoveL Offs(pOrigin,184.39,106.04,0.00),v40,z0,tPen\WObj:=wPaper;
    MoveL Offs(pOrigin,183.92,105.56,0.00),v40,z0,tPen\WObj:=wPaper;
    MoveL Offs(pOrigin,183.92,106.04,0.00),v40,z0,tPen\WObj:=wPaper;
    MoveL Offs(pOrigin,184.39,106.04,0.00),v40,fine,tPen\WObj:=wPaper;
    MoveL Offs(pOrigin,184.39,106.04,6.00),v60,z5,tPen\WObj:=wPaper;
    MoveL Offs(pOrigin,182.96,104.13,6.00),vTravel,z5,tPen\WObj:=wPaper;
    MoveL Offs(pOrigin,182.96,104.13,0.00),v60,z0,tPen\WObj:=wPaper;
    MoveL Offs(pOrigin,182.48,103.65,0.00),v40,z0,tPen\WObj:=wPaper;
    MoveL Offs(pOrigin,182.48,104.13,0.00),v40,z0,tPen\WObj:=wPaper;
    MoveL Offs(pOrigin,182.96,104.13,0.00),v40,z0,tPen\WObj:=wPaper;
    MoveL Offs(pOrigin,182.48,103.65,0.00),v40,z0,tPen\WObj:=wPaper;
    MoveL Offs(pOrigin,182.48,104.13,0.00),v40,z0,tPen\WObj:=wPaper;
    MoveL Offs(pOrigin,182.96,104.13,0.00),v40,fine,tPen\WObj:=wPaper;
    MoveL Offs(pOrigin,182.96,104.13,6.00),v60,z5,tPen\WObj:=wPaper;
    MoveL Offs(pOrigin,182.00,102.69,6.00),vTravel,z5,tPen\WObj:=wPaper;
    MoveL Offs(pOrigin,182.00,102.69,0.00),v60,z0,tPen\WObj:=wPaper;
    MoveL Offs(pOrigin,181.04,101.73,0.00),v40,z0,tPen\WObj:=wPaper;
    MoveL Offs(pOrigin,181.04,102.21,0.00),v40,z0,tPen\WObj:=wPaper;
    MoveL Offs(pOrigin,181.52,102.21,0.00),v40,z0,tPen\WObj:=wPaper;
    MoveL Offs(pOrigin,182.00,102.69,0.00),v40,z0,tPen\WObj:=wPaper;
    MoveL Offs(pOrigin,181.04,101.73,0.00),v40,z0,tPen\WObj:=wPaper;
    MoveL Offs(pOrigin,181.04,102.21,0.00),v40,z0,tPen\WObj:=wPaper;
    MoveL Offs(pOrigin,181.52,102.21,0.00),v40,z0,tPen\WObj:=wPaper;
    MoveL Offs(pOrigin,182.00,102.69,0.00),v40,fine,tPen\WObj:=wPaper;
    MoveL Offs(pOrigin,182.00,102.69,6.00),v60,z5,tPen\WObj:=wPaper;
    MoveL Offs(pOrigin,180.08,100.30,6.00),vTravel,z5,tPen\WObj:=wPaper;
    MoveL Offs(pOrigin,180.08,100.30,0.00),v60,z0,tPen\WObj:=wPaper;
    MoveL Offs(pOrigin,178.65,98.86,0.00),v40,z0,tPen\WObj:=wPaper;
    MoveL Offs(pOrigin,178.65,99.34,0.00),v40,z0,tPen\WObj:=wPaper;
    MoveL Offs(pOrigin,179.13,99.34,0.00),v40,z0,tPen\WObj:=wPaper;
    MoveL Offs(pOrigin,180.08,100.30,0.00),v40,z0,tPen\WObj:=wPaper;
    MoveL Offs(pOrigin,178.65,98.86,0.00),v40,z0,tPen\WObj:=wPaper;
    MoveL Offs(pOrigin,178.65,99.34,0.00),v40,z0,tPen\WObj:=wPaper;
    MoveL Offs(pOrigin,179.13,99.34,0.00),v40,z0,tPen\WObj:=wPaper;
    MoveL Offs(pOrigin,180.08,100.30,0.00),v40,fine,tPen\WObj:=wPaper;
    MoveL Offs(pOrigin,180.08,100.30,6.00),v60,z5,tPen\WObj:=wPaper;
    MoveL Offs(pOrigin,176.73,96.46,6.00),vTravel,z5,tPen\WObj:=wPaper;
    MoveL Offs(pOrigin,176.73,96.46,0.00),v60,z0,tPen\WObj:=wPaper;
    MoveL Offs(pOrigin,176.25,95.99,0.00),v40,z0,tPen\WObj:=wPaper;
    MoveL Offs(pOrigin,176.25,96.46,0.00),v40,z0,tPen\WObj:=wPaper;
    MoveL Offs(pOrigin,176.73,96.46,0.00),v40,z0,tPen\WObj:=wPaper;
    MoveL Offs(pOrigin,176.25,95.99,0.00),v40,z0,tPen\WObj:=wPaper;
    MoveL Offs(pOrigin,176.25,96.46,0.00),v40,z0,tPen\WObj:=wPaper;
    MoveL Offs(pOrigin,176.73,96.46,0.00),v40,fine,tPen\WObj:=wPaper;
    MoveL Offs(pOrigin,176.73,96.46,6.00),v60,z5,tPen\WObj:=wPaper;
    MoveL Offs(pOrigin,170.67,90.56,6.00),vTravel,z5,tPen\WObj:=wPaper;
    MoveL Offs(pOrigin,170.67,90.56,0.00),v60,z0,tPen\WObj:=wPaper;
    MoveL Offs(pOrigin,175.30,95.03,0.00),v40,z0,tPen\WObj:=wPaper;
    MoveL Offs(pOrigin,170.67,90.56,0.00),v40,fine,tPen\WObj:=wPaper;
    MoveL Offs(pOrigin,170.67,90.56,6.00),v60,z5,tPen\WObj:=wPaper;
    MoveL Offs(pOrigin,169.55,89.76,6.00),vTravel,z5,tPen\WObj:=wPaper;
    MoveL Offs(pOrigin,169.55,89.76,0.00),v60,z0,tPen\WObj:=wPaper;
    MoveL Offs(pOrigin,166.68,86.89,0.00),v40,z0,tPen\WObj:=wPaper;
    MoveL Offs(pOrigin,166.68,87.37,0.00),v40,z0,tPen\WObj:=wPaper;
    MoveL Offs(pOrigin,167.15,87.37,0.00),v40,z0,tPen\WObj:=wPaper;
    MoveL Offs(pOrigin,169.55,89.76,0.00),v40,z0,tPen\WObj:=wPaper;
    MoveL Offs(pOrigin,166.68,86.89,0.00),v40,z0,tPen\WObj:=wPaper;
    MoveL Offs(pOrigin,166.68,87.37,0.00),v40,z0,tPen\WObj:=wPaper;
    MoveL Offs(pOrigin,167.15,87.37,0.00),v40,z0,tPen\WObj:=wPaper;
    MoveL Offs(pOrigin,169.55,89.76,0.00),v40,fine,tPen\WObj:=wPaper;
    MoveL Offs(pOrigin,169.55,89.76,6.00),v60,z5,tPen\WObj:=wPaper;
    MoveL Offs(pOrigin,165.72,86.41,6.00),vTravel,z5,tPen\WObj:=wPaper;
    MoveL Offs(pOrigin,165.72,86.41,0.00),v60,z0,tPen\WObj:=wPaper;
    MoveL Offs(pOrigin,165.24,85.93,0.00),v40,z0,tPen\WObj:=wPaper;
    MoveL Offs(pOrigin,165.24,86.41,0.00),v40,z0,tPen\WObj:=wPaper;
    MoveL Offs(pOrigin,165.72,86.41,0.00),v40,z0,tPen\WObj:=wPaper;
    MoveL Offs(pOrigin,165.24,85.93,0.00),v40,z0,tPen\WObj:=wPaper;
    MoveL Offs(pOrigin,165.24,86.41,0.00),v40,z0,tPen\WObj:=wPaper;
    MoveL Offs(pOrigin,165.72,86.41,0.00),v40,fine,tPen\WObj:=wPaper;
    MoveL Offs(pOrigin,165.72,86.41,6.00),v60,z5,tPen\WObj:=wPaper;
    MoveL Offs(pOrigin,164.28,85.45,6.00),vTravel,z5,tPen\WObj:=wPaper;
    MoveL Offs(pOrigin,164.28,85.45,0.00),v60,z0,tPen\WObj:=wPaper;
    MoveL Offs(pOrigin,163.32,84.49,0.00),v40,z0,tPen\WObj:=wPaper;
  ENDPROC

  PROC DrawPart5()
    MoveL Offs(pOrigin,163.32,84.97,0.00),v40,z0,tPen\WObj:=wPaper;
    MoveL Offs(pOrigin,163.80,84.97,0.00),v40,z0,tPen\WObj:=wPaper;
    MoveL Offs(pOrigin,164.28,85.45,0.00),v40,z0,tPen\WObj:=wPaper;
    MoveL Offs(pOrigin,163.32,84.49,0.00),v40,z0,tPen\WObj:=wPaper;
    MoveL Offs(pOrigin,163.32,84.97,0.00),v40,z0,tPen\WObj:=wPaper;
    MoveL Offs(pOrigin,163.80,84.97,0.00),v40,z0,tPen\WObj:=wPaper;
    MoveL Offs(pOrigin,164.28,85.45,0.00),v40,fine,tPen\WObj:=wPaper;
    MoveL Offs(pOrigin,164.28,85.45,6.00),v60,z5,tPen\WObj:=wPaper;
    MoveL Offs(pOrigin,162.37,84.01,6.00),vTravel,z5,tPen\WObj:=wPaper;
    MoveL Offs(pOrigin,162.37,84.01,0.00),v60,z0,tPen\WObj:=wPaper;
    MoveL Offs(pOrigin,161.89,83.54,0.00),v40,z0,tPen\WObj:=wPaper;
    MoveL Offs(pOrigin,161.89,84.01,0.00),v40,z0,tPen\WObj:=wPaper;
    MoveL Offs(pOrigin,162.37,84.01,0.00),v40,z0,tPen\WObj:=wPaper;
    MoveL Offs(pOrigin,161.89,83.54,0.00),v40,z0,tPen\WObj:=wPaper;
    MoveL Offs(pOrigin,161.89,84.01,0.00),v40,z0,tPen\WObj:=wPaper;
    MoveL Offs(pOrigin,162.37,84.01,0.00),v40,fine,tPen\WObj:=wPaper;
    MoveL Offs(pOrigin,162.37,84.01,6.00),v60,z5,tPen\WObj:=wPaper;
    MoveL Offs(pOrigin,159.97,82.58,6.00),vTravel,z5,tPen\WObj:=wPaper;
    MoveL Offs(pOrigin,159.97,82.58,0.00),v60,z0,tPen\WObj:=wPaper;
    MoveL Offs(pOrigin,159.49,82.10,0.00),v40,z0,tPen\WObj:=wPaper;
    MoveL Offs(pOrigin,159.49,82.58,0.00),v40,z0,tPen\WObj:=wPaper;
    MoveL Offs(pOrigin,159.97,82.58,0.00),v40,z0,tPen\WObj:=wPaper;
    MoveL Offs(pOrigin,159.49,82.10,0.00),v40,z0,tPen\WObj:=wPaper;
    MoveL Offs(pOrigin,159.49,82.58,0.00),v40,z0,tPen\WObj:=wPaper;
    MoveL Offs(pOrigin,159.97,82.58,0.00),v40,fine,tPen\WObj:=wPaper;
    MoveL Offs(pOrigin,159.97,82.58,6.00),v60,z5,tPen\WObj:=wPaper;
    MoveL Offs(pOrigin,182.00,82.10,6.00),vTravel,z5,tPen\WObj:=wPaper;
    MoveL Offs(pOrigin,182.00,82.10,0.00),v60,z0,tPen\WObj:=wPaper;
    MoveL Offs(pOrigin,182.48,81.62,0.00),v40,z0,tPen\WObj:=wPaper;
    MoveL Offs(pOrigin,182.96,81.62,0.00),v40,z0,tPen\WObj:=wPaper;
    MoveL Offs(pOrigin,183.44,81.14,0.00),v40,z0,tPen\WObj:=wPaper;
    MoveL Offs(pOrigin,183.44,80.66,0.00),v40,z0,tPen\WObj:=wPaper;
    MoveL Offs(pOrigin,182.96,81.14,0.00),v40,z0,tPen\WObj:=wPaper;
    MoveL Offs(pOrigin,182.96,84.01,0.00),v40,z0,tPen\WObj:=wPaper;
    MoveL Offs(pOrigin,182.48,83.54,0.00),v40,z0,tPen\WObj:=wPaper;
    MoveL Offs(pOrigin,182.00,82.10,0.00),v40,z0,tPen\WObj:=wPaper;
    MoveL Offs(pOrigin,182.48,81.62,0.00),v40,z0,tPen\WObj:=wPaper;
    MoveL Offs(pOrigin,182.96,81.62,0.00),v40,z0,tPen\WObj:=wPaper;
    MoveL Offs(pOrigin,183.44,81.14,0.00),v40,z0,tPen\WObj:=wPaper;
    MoveL Offs(pOrigin,183.44,80.66,0.00),v40,z0,tPen\WObj:=wPaper;
    MoveL Offs(pOrigin,182.96,81.14,0.00),v40,z0,tPen\WObj:=wPaper;
    MoveL Offs(pOrigin,182.96,84.01,0.00),v40,z0,tPen\WObj:=wPaper;
    MoveL Offs(pOrigin,182.48,83.54,0.00),v40,z0,tPen\WObj:=wPaper;
    MoveL Offs(pOrigin,182.00,82.10,0.00),v40,fine,tPen\WObj:=wPaper;
    MoveL Offs(pOrigin,182.00,82.10,6.00),v60,z5,tPen\WObj:=wPaper;
    MoveL Offs(pOrigin,184.39,80.50,6.00),vTravel,z5,tPen\WObj:=wPaper;
    MoveL Offs(pOrigin,184.39,80.50,0.00),v60,z0,tPen\WObj:=wPaper;
    MoveL Offs(pOrigin,192.54,76.03,0.00),v40,z0,tPen\WObj:=wPaper;
    MoveL Offs(pOrigin,193.33,75.23,0.00),v40,z0,tPen\WObj:=wPaper;
    MoveL Offs(pOrigin,184.39,80.50,0.00),v40,fine,tPen\WObj:=wPaper;
    MoveL Offs(pOrigin,184.39,80.50,6.00),v60,z5,tPen\WObj:=wPaper;
    MoveL Offs(pOrigin,184.39,84.49,6.00),vTravel,z5,tPen\WObj:=wPaper;
    MoveL Offs(pOrigin,184.39,84.49,0.00),v60,z0,tPen\WObj:=wPaper;
    MoveL Offs(pOrigin,184.39,84.97,0.00),v40,z0,tPen\WObj:=wPaper;
    MoveL Offs(pOrigin,184.87,84.97,0.00),v40,z0,tPen\WObj:=wPaper;
    MoveL Offs(pOrigin,184.39,84.49,0.00),v40,z0,tPen\WObj:=wPaper;
    MoveL Offs(pOrigin,184.39,84.97,0.00),v40,z0,tPen\WObj:=wPaper;
    MoveL Offs(pOrigin,184.87,84.97,0.00),v40,z0,tPen\WObj:=wPaper;
    MoveL Offs(pOrigin,184.39,84.49,0.00),v40,z0,tPen\WObj:=wPaper;
    MoveL Offs(pOrigin,183.92,84.49,0.00),v40,z0,tPen\WObj:=wPaper;
    MoveL Offs(pOrigin,186.31,86.09,0.00),v40,z0,tPen\WObj:=wPaper;
    MoveL Offs(pOrigin,188.23,86.41,0.00),v40,z0,tPen\WObj:=wPaper;
    MoveL Offs(pOrigin,192.69,84.17,0.00),v40,z0,tPen\WObj:=wPaper;
    MoveL Offs(pOrigin,189.66,84.01,0.00),v40,z0,tPen\WObj:=wPaper;
    MoveL Offs(pOrigin,183.92,84.49,0.00),v40,fine,tPen\WObj:=wPaper;
    MoveL Offs(pOrigin,183.92,84.49,6.00),v60,z5,tPen\WObj:=wPaper;
    MoveL Offs(pOrigin,193.65,83.54,6.00),vTravel,z5,tPen\WObj:=wPaper;
    MoveL Offs(pOrigin,193.65,83.54,0.00),v60,z0,tPen\WObj:=wPaper;
    MoveL Offs(pOrigin,283.04,68.85,0.00),v40,z0,tPen\WObj:=wPaper;
    MoveL Offs(pOrigin,296.45,73.80,0.00),v40,z0,tPen\WObj:=wPaper;
    MoveL Offs(pOrigin,307.94,79.54,0.00),v40,z0,tPen\WObj:=wPaper;
    MoveL Offs(pOrigin,317.52,85.45,0.00),v40,z0,tPen\WObj:=wPaper;
    MoveL Offs(pOrigin,322.79,89.28,0.00),v40,z0,tPen\WObj:=wPaper;
    MoveL Offs(pOrigin,330.93,95.99,0.00),v40,z0,tPen\WObj:=wPaper;
    MoveL Offs(pOrigin,341.46,106.52,0.00),v40,z0,tPen\WObj:=wPaper;
    MoveL Offs(pOrigin,349.61,117.06,0.00),v40,z0,tPen\WObj:=wPaper;
    MoveL Offs(pOrigin,354.08,123.76,0.00),v40,z0,tPen\WObj:=wPaper;
    MoveL Offs(pOrigin,359.50,133.34,0.00),v40,z0,tPen\WObj:=wPaper;
    MoveL Offs(pOrigin,364.13,143.39,0.00),v40,z0,tPen\WObj:=wPaper;
    MoveL Offs(pOrigin,367.80,153.93,0.00),v40,z0,tPen\WObj:=wPaper;
    MoveL Offs(pOrigin,369.24,159.20,0.00),v40,z0,tPen\WObj:=wPaper;
    MoveL Offs(pOrigin,369.24,160.15,0.00),v40,z0,tPen\WObj:=wPaper;
    MoveL Offs(pOrigin,368.76,160.79,0.00),v40,z0,tPen\WObj:=wPaper;
    MoveL Offs(pOrigin,367.80,160.63,0.00),v40,z0,tPen\WObj:=wPaper;
    MoveL Offs(pOrigin,359.66,152.97,0.00),v40,z0,tPen\WObj:=wPaper;
    MoveL Offs(pOrigin,355.03,141.48,0.00),v40,z0,tPen\WObj:=wPaper;
    MoveL Offs(pOrigin,349.29,130.46,0.00),v40,z0,tPen\WObj:=wPaper;
    MoveL Offs(pOrigin,343.86,121.85,0.00),v40,z0,tPen\WObj:=wPaper;
    MoveL Offs(pOrigin,335.24,110.83,0.00),v40,z0,tPen\WObj:=wPaper;
    MoveL Offs(pOrigin,325.66,101.25,0.00),v40,z0,tPen\WObj:=wPaper;
    MoveL Offs(pOrigin,315.13,93.11,0.00),v40,z0,tPen\WObj:=wPaper;
    MoveL Offs(pOrigin,305.55,87.05,0.00),v40,z0,tPen\WObj:=wPaper;
    MoveL Offs(pOrigin,301.24,84.65,0.00),v40,z0,tPen\WObj:=wPaper;
    MoveL Offs(pOrigin,293.10,80.82,0.00),v40,z0,tPen\WObj:=wPaper;
    MoveL Offs(pOrigin,288.79,79.07,0.00),v40,z0,tPen\WObj:=wPaper;
    MoveL Offs(pOrigin,285.44,78.11,0.00),v40,z0,tPen\WObj:=wPaper;
    MoveL Offs(pOrigin,284.48,77.47,0.00),v40,z0,tPen\WObj:=wPaper;
    MoveL Offs(pOrigin,276.34,74.92,0.00),v40,z0,tPen\WObj:=wPaper;
    MoveL Offs(pOrigin,273.46,74.44,0.00),v40,z0,tPen\WObj:=wPaper;
    MoveL Offs(pOrigin,270.59,73.48,0.00),v40,z0,tPen\WObj:=wPaper;
    MoveL Offs(pOrigin,268.68,73.48,0.00),v40,z0,tPen\WObj:=wPaper;
    MoveL Offs(pOrigin,265.80,72.52,0.00),v40,z0,tPen\WObj:=wPaper;
    MoveL Offs(pOrigin,264.37,72.52,0.00),v40,z0,tPen\WObj:=wPaper;
    MoveL Offs(pOrigin,262.93,72.04,0.00),v40,z0,tPen\WObj:=wPaper;
    MoveL Offs(pOrigin,260.06,72.04,0.00),v40,z0,tPen\WObj:=wPaper;
    MoveL Offs(pOrigin,257.18,71.08,0.00),v40,z0,tPen\WObj:=wPaper;
    MoveL Offs(pOrigin,232.76,71.08,0.00),v40,z0,tPen\WObj:=wPaper;
    MoveL Offs(pOrigin,228.93,72.04,0.00),v40,z0,tPen\WObj:=wPaper;
    MoveL Offs(pOrigin,224.14,72.52,0.00),v40,z0,tPen\WObj:=wPaper;
    MoveL Offs(pOrigin,221.27,73.48,0.00),v40,z0,tPen\WObj:=wPaper;
    MoveL Offs(pOrigin,219.83,73.48,0.00),v40,z0,tPen\WObj:=wPaper;
    MoveL Offs(pOrigin,211.69,75.87,0.00),v40,z0,tPen\WObj:=wPaper;
    MoveL Offs(pOrigin,202.59,79.07,0.00),v40,z0,tPen\WObj:=wPaper;
    MoveL Offs(pOrigin,197.32,81.78,0.00),v40,z0,tPen\WObj:=wPaper;
    MoveL Offs(pOrigin,195.41,82.42,0.00),v40,z0,tPen\WObj:=wPaper;
    MoveL Offs(pOrigin,193.65,83.54,0.00),v40,fine,tPen\WObj:=wPaper;
    MoveL Offs(pOrigin,193.65,83.54,6.00),v60,z5,tPen\WObj:=wPaper;
    MoveL Offs(pOrigin,194.45,74.76,6.00),vTravel,z5,tPen\WObj:=wPaper;
    MoveL Offs(pOrigin,194.45,74.76,0.00),v60,z0,tPen\WObj:=wPaper;
    MoveL Offs(pOrigin,202.11,71.40,0.00),v40,z0,tPen\WObj:=wPaper;
  ENDPROC

  PROC DrawPart6()
    MoveL Offs(pOrigin,207.86,69.49,0.00),v40,z0,tPen\WObj:=wPaper;
    MoveL Offs(pOrigin,208.82,68.85,0.00),v40,z0,tPen\WObj:=wPaper;
    MoveL Offs(pOrigin,216.96,66.30,0.00),v40,z0,tPen\WObj:=wPaper;
    MoveL Offs(pOrigin,218.39,66.30,0.00),v40,z0,tPen\WObj:=wPaper;
    MoveL Offs(pOrigin,221.27,65.34,0.00),v40,z0,tPen\WObj:=wPaper;
    MoveL Offs(pOrigin,222.70,65.34,0.00),v40,z0,tPen\WObj:=wPaper;
    MoveL Offs(pOrigin,228.93,63.90,0.00),v40,z0,tPen\WObj:=wPaper;
    MoveL Offs(pOrigin,233.72,63.90,0.00),v40,z0,tPen\WObj:=wPaper;
    MoveL Offs(pOrigin,238.03,62.94,0.00),v40,z0,tPen\WObj:=wPaper;
    MoveL Offs(pOrigin,251.44,62.94,0.00),v40,z0,tPen\WObj:=wPaper;
    MoveL Offs(pOrigin,252.87,63.42,0.00),v40,z0,tPen\WObj:=wPaper;
    MoveL Offs(pOrigin,255.27,63.42,0.00),v40,z0,tPen\WObj:=wPaper;
    MoveL Offs(pOrigin,256.70,63.90,0.00),v40,z0,tPen\WObj:=wPaper;
    MoveL Offs(pOrigin,261.49,63.90,0.00),v40,z0,tPen\WObj:=wPaper;
    MoveL Offs(pOrigin,265.32,64.86,0.00),v40,z0,tPen\WObj:=wPaper;
    MoveL Offs(pOrigin,267.24,64.86,0.00),v40,z0,tPen\WObj:=wPaper;
    MoveL Offs(pOrigin,272.99,66.30,0.00),v40,z0,tPen\WObj:=wPaper;
    MoveL Offs(pOrigin,274.42,66.30,0.00),v40,z0,tPen\WObj:=wPaper;
    MoveL Offs(pOrigin,281.61,68.53,0.00),v40,z0,tPen\WObj:=wPaper;
    MoveL Offs(pOrigin,194.45,74.76,0.00),v40,fine,tPen\WObj:=wPaper;
    MoveL Offs(pOrigin,194.45,74.76,6.00),v60,z5,tPen\WObj:=wPaper;
    MoveL Offs(pOrigin,204.03,93.11,6.00),vTravel,z5,tPen\WObj:=wPaper;
    MoveL Offs(pOrigin,204.03,93.11,0.00),v60,z0,tPen\WObj:=wPaper;
    MoveL Offs(pOrigin,203.23,93.59,0.00),v40,z0,tPen\WObj:=wPaper;
    MoveL Offs(pOrigin,313.69,127.59,0.00),v40,z0,tPen\WObj:=wPaper;
    MoveL Offs(pOrigin,320.87,127.59,0.00),v40,z0,tPen\WObj:=wPaper;
    MoveL Offs(pOrigin,322.31,128.07,0.00),v40,z0,tPen\WObj:=wPaper;
    MoveL Offs(pOrigin,329.01,128.07,0.00),v40,z0,tPen\WObj:=wPaper;
    MoveL Offs(pOrigin,330.93,127.43,0.00),v40,z0,tPen\WObj:=wPaper;
    MoveL Offs(pOrigin,331.41,126.63,0.00),v40,z0,tPen\WObj:=wPaper;
    MoveL Offs(pOrigin,331.09,124.72,0.00),v40,z0,tPen\WObj:=wPaper;
    MoveL Offs(pOrigin,330.45,123.92,0.00),v40,z0,tPen\WObj:=wPaper;
    MoveL Offs(pOrigin,326.14,122.32,0.00),v40,z0,tPen\WObj:=wPaper;
    MoveL Offs(pOrigin,325.18,122.32,0.00),v40,z0,tPen\WObj:=wPaper;
    MoveL Offs(pOrigin,322.31,121.37,0.00),v40,z0,tPen\WObj:=wPaper;
    MoveL Offs(pOrigin,320.39,121.37,0.00),v40,z0,tPen\WObj:=wPaper;
    MoveL Offs(pOrigin,315.13,119.93,0.00),v40,z0,tPen\WObj:=wPaper;
    MoveL Offs(pOrigin,313.69,119.93,0.00),v40,z0,tPen\WObj:=wPaper;
    MoveL Offs(pOrigin,310.82,118.97,0.00),v40,z0,tPen\WObj:=wPaper;
    MoveL Offs(pOrigin,307.94,118.97,0.00),v40,z0,tPen\WObj:=wPaper;
    MoveL Offs(pOrigin,302.68,117.54,0.00),v40,z0,tPen\WObj:=wPaper;
    MoveL Offs(pOrigin,300.76,117.54,0.00),v40,z0,tPen\WObj:=wPaper;
    MoveL Offs(pOrigin,293.58,115.62,0.00),v40,z0,tPen\WObj:=wPaper;
    MoveL Offs(pOrigin,289.75,115.14,0.00),v40,z0,tPen\WObj:=wPaper;
    MoveL Offs(pOrigin,286.87,114.18,0.00),v40,z0,tPen\WObj:=wPaper;
    MoveL Offs(pOrigin,284.96,114.18,0.00),v40,z0,tPen\WObj:=wPaper;
    MoveL Offs(pOrigin,275.86,111.79,0.00),v40,z0,tPen\WObj:=wPaper;
    MoveL Offs(pOrigin,274.42,111.79,0.00),v40,z0,tPen\WObj:=wPaper;
    MoveL Offs(pOrigin,269.15,110.35,0.00),v40,z0,tPen\WObj:=wPaper;
    MoveL Offs(pOrigin,268.20,110.35,0.00),v40,z0,tPen\WObj:=wPaper;
    MoveL Offs(pOrigin,265.80,109.39,0.00),v40,z0,tPen\WObj:=wPaper;
    MoveL Offs(pOrigin,264.37,109.39,0.00),v40,z0,tPen\WObj:=wPaper;
    MoveL Offs(pOrigin,246.65,104.61,0.00),v40,z0,tPen\WObj:=wPaper;
    MoveL Offs(pOrigin,245.69,104.61,0.00),v40,z0,tPen\WObj:=wPaper;
    MoveL Offs(pOrigin,241.38,103.17,0.00),v40,z0,tPen\WObj:=wPaper;
    MoveL Offs(pOrigin,240.42,103.17,0.00),v40,z0,tPen\WObj:=wPaper;
    MoveL Offs(pOrigin,238.03,102.21,0.00),v40,z0,tPen\WObj:=wPaper;
    MoveL Offs(pOrigin,237.07,102.21,0.00),v40,z0,tPen\WObj:=wPaper;
    MoveL Offs(pOrigin,229.41,99.82,0.00),v40,z0,tPen\WObj:=wPaper;
    MoveL Offs(pOrigin,228.45,99.82,0.00),v40,z0,tPen\WObj:=wPaper;
    MoveL Offs(pOrigin,208.82,94.07,0.00),v40,z0,tPen\WObj:=wPaper;
    MoveL Offs(pOrigin,204.99,93.11,0.00),v40,z0,tPen\WObj:=wPaper;
    MoveL Offs(pOrigin,204.03,93.11,0.00),v40,fine,tPen\WObj:=wPaper;
    MoveL Offs(pOrigin,204.03,93.11,6.00),v60,z5,tPen\WObj:=wPaper;
    MoveL Offs(pOrigin,202.59,94.07,6.00),vTravel,z5,tPen\WObj:=wPaper;
    MoveL Offs(pOrigin,202.59,94.07,0.00),v60,z0,tPen\WObj:=wPaper;
    MoveL Offs(pOrigin,202.11,94.07,0.00),v40,z0,tPen\WObj:=wPaper;
    MoveL Offs(pOrigin,201.63,94.55,0.00),v40,z0,tPen\WObj:=wPaper;
    MoveL Offs(pOrigin,202.11,94.55,0.00),v40,z0,tPen\WObj:=wPaper;
    MoveL Offs(pOrigin,202.59,94.07,0.00),v40,z0,tPen\WObj:=wPaper;
    MoveL Offs(pOrigin,202.11,94.07,0.00),v40,z0,tPen\WObj:=wPaper;
    MoveL Offs(pOrigin,201.63,94.55,0.00),v40,z0,tPen\WObj:=wPaper;
    MoveL Offs(pOrigin,202.11,94.55,0.00),v40,z0,tPen\WObj:=wPaper;
    MoveL Offs(pOrigin,202.59,94.07,0.00),v40,fine,tPen\WObj:=wPaper;
    MoveL Offs(pOrigin,202.59,94.07,6.00),v60,z5,tPen\WObj:=wPaper;
    MoveL Offs(pOrigin,201.63,95.51,6.00),vTravel,z5,tPen\WObj:=wPaper;
    MoveL Offs(pOrigin,201.63,95.51,0.00),v60,z0,tPen\WObj:=wPaper;
    MoveL Offs(pOrigin,201.79,96.46,0.00),v40,z0,tPen\WObj:=wPaper;
    MoveL Offs(pOrigin,206.74,104.61,0.00),v40,z0,tPen\WObj:=wPaper;
    MoveL Offs(pOrigin,210.25,109.87,0.00),v40,z0,tPen\WObj:=wPaper;
    MoveL Offs(pOrigin,211.69,110.99,0.00),v40,z0,tPen\WObj:=wPaper;
    MoveL Offs(pOrigin,228.93,115.62,0.00),v40,z0,tPen\WObj:=wPaper;
    MoveL Offs(pOrigin,230.37,115.62,0.00),v40,z0,tPen\WObj:=wPaper;
    MoveL Offs(pOrigin,237.55,117.54,0.00),v40,z0,tPen\WObj:=wPaper;
    MoveL Offs(pOrigin,241.38,118.01,0.00),v40,z0,tPen\WObj:=wPaper;
    MoveL Offs(pOrigin,243.77,118.97,0.00),v40,z0,tPen\WObj:=wPaper;
    MoveL Offs(pOrigin,246.17,118.97,0.00),v40,z0,tPen\WObj:=wPaper;
    MoveL Offs(pOrigin,251.92,120.41,0.00),v40,z0,tPen\WObj:=wPaper;
    MoveL Offs(pOrigin,254.31,120.41,0.00),v40,z0,tPen\WObj:=wPaper;
    MoveL Offs(pOrigin,257.66,121.37,0.00),v40,z0,tPen\WObj:=wPaper;
    MoveL Offs(pOrigin,260.06,121.37,0.00),v40,z0,tPen\WObj:=wPaper;
    MoveL Offs(pOrigin,263.89,122.32,0.00),v40,z0,tPen\WObj:=wPaper;
    MoveL Offs(pOrigin,265.80,122.32,0.00),v40,z0,tPen\WObj:=wPaper;
    MoveL Offs(pOrigin,267.24,122.80,0.00),v40,z0,tPen\WObj:=wPaper;
    MoveL Offs(pOrigin,270.11,122.80,0.00),v40,z0,tPen\WObj:=wPaper;
    MoveL Offs(pOrigin,273.46,123.76,0.00),v40,z0,tPen\WObj:=wPaper;
    MoveL Offs(pOrigin,277.77,123.76,0.00),v40,z0,tPen\WObj:=wPaper;
    MoveL Offs(pOrigin,279.21,124.24,0.00),v40,z0,tPen\WObj:=wPaper;
    MoveL Offs(pOrigin,281.61,124.40,0.00),v40,z0,tPen\WObj:=wPaper;
    MoveL Offs(pOrigin,201.63,95.51,0.00),v40,fine,tPen\WObj:=wPaper;
    MoveL Offs(pOrigin,201.63,95.51,6.00),v60,z5,tPen\WObj:=wPaper;
    MoveL Offs(pOrigin,202.59,96.94,6.00),vTravel,z5,tPen\WObj:=wPaper;
    MoveL Offs(pOrigin,202.59,96.94,0.00),v60,z0,tPen\WObj:=wPaper;
    MoveL Offs(pOrigin,202.59,97.42,0.00),v40,z0,tPen\WObj:=wPaper;
    MoveL Offs(pOrigin,203.07,97.90,0.00),v40,z0,tPen\WObj:=wPaper;
    MoveL Offs(pOrigin,202.59,96.94,0.00),v40,z0,tPen\WObj:=wPaper;
    MoveL Offs(pOrigin,202.59,97.42,0.00),v40,z0,tPen\WObj:=wPaper;
    MoveL Offs(pOrigin,203.07,97.90,0.00),v40,z0,tPen\WObj:=wPaper;
    MoveL Offs(pOrigin,202.59,96.94,0.00),v40,fine,tPen\WObj:=wPaper;
    MoveL Offs(pOrigin,202.59,96.94,6.00),v60,z5,tPen\WObj:=wPaper;
    MoveL Offs(pOrigin,203.55,98.38,6.00),vTravel,z5,tPen\WObj:=wPaper;
    MoveL Offs(pOrigin,203.55,98.38,0.00),v60,z0,tPen\WObj:=wPaper;
    MoveL Offs(pOrigin,203.55,98.86,0.00),v40,z0,tPen\WObj:=wPaper;
    MoveL Offs(pOrigin,204.03,99.34,0.00),v40,z0,tPen\WObj:=wPaper;
    MoveL Offs(pOrigin,203.55,98.38,0.00),v40,z0,tPen\WObj:=wPaper;
    MoveL Offs(pOrigin,203.55,98.86,0.00),v40,z0,tPen\WObj:=wPaper;
    MoveL Offs(pOrigin,204.03,99.34,0.00),v40,z0,tPen\WObj:=wPaper;
    MoveL Offs(pOrigin,203.55,98.38,0.00),v40,fine,tPen\WObj:=wPaper;
    MoveL Offs(pOrigin,203.55,98.38,6.00),v60,z5,tPen\WObj:=wPaper;
    MoveL Offs(pOrigin,204.51,100.30,6.00),vTravel,z5,tPen\WObj:=wPaper;
  ENDPROC

  PROC DrawPart7()
    MoveL Offs(pOrigin,204.51,100.30,0.00),v60,z0,tPen\WObj:=wPaper;
    MoveL Offs(pOrigin,204.51,100.77,0.00),v40,z0,tPen\WObj:=wPaper;
    MoveL Offs(pOrigin,204.99,100.77,0.00),v40,z0,tPen\WObj:=wPaper;
    MoveL Offs(pOrigin,204.51,100.30,0.00),v40,z0,tPen\WObj:=wPaper;
    MoveL Offs(pOrigin,204.51,100.77,0.00),v40,z0,tPen\WObj:=wPaper;
    MoveL Offs(pOrigin,204.99,100.77,0.00),v40,z0,tPen\WObj:=wPaper;
    MoveL Offs(pOrigin,204.51,100.30,0.00),v40,fine,tPen\WObj:=wPaper;
    MoveL Offs(pOrigin,204.51,100.30,6.00),v60,z5,tPen\WObj:=wPaper;
    MoveL Offs(pOrigin,205.94,102.69,6.00),vTravel,z5,tPen\WObj:=wPaper;
    MoveL Offs(pOrigin,205.94,102.69,0.00),v60,z0,tPen\WObj:=wPaper;
    MoveL Offs(pOrigin,205.94,103.17,0.00),v40,z0,tPen\WObj:=wPaper;
    MoveL Offs(pOrigin,206.42,103.17,0.00),v40,z0,tPen\WObj:=wPaper;
    MoveL Offs(pOrigin,205.94,102.69,0.00),v40,z0,tPen\WObj:=wPaper;
    MoveL Offs(pOrigin,205.94,103.17,0.00),v40,z0,tPen\WObj:=wPaper;
    MoveL Offs(pOrigin,206.42,103.17,0.00),v40,z0,tPen\WObj:=wPaper;
    MoveL Offs(pOrigin,205.94,102.69,0.00),v40,fine,tPen\WObj:=wPaper;
    MoveL Offs(pOrigin,205.94,102.69,6.00),v60,z5,tPen\WObj:=wPaper;
    MoveL Offs(pOrigin,206.90,104.13,6.00),vTravel,z5,tPen\WObj:=wPaper;
    MoveL Offs(pOrigin,206.90,104.13,0.00),v60,z0,tPen\WObj:=wPaper;
    MoveL Offs(pOrigin,206.90,104.61,0.00),v40,z0,tPen\WObj:=wPaper;
    MoveL Offs(pOrigin,208.34,106.04,0.00),v40,z0,tPen\WObj:=wPaper;
    MoveL Offs(pOrigin,206.90,104.13,0.00),v40,z0,tPen\WObj:=wPaper;
    MoveL Offs(pOrigin,206.90,104.61,0.00),v40,z0,tPen\WObj:=wPaper;
    MoveL Offs(pOrigin,208.34,106.04,0.00),v40,z0,tPen\WObj:=wPaper;
    MoveL Offs(pOrigin,206.90,104.13,0.00),v40,fine,tPen\WObj:=wPaper;
    MoveL Offs(pOrigin,206.90,104.13,6.00),v60,z5,tPen\WObj:=wPaper;
    MoveL Offs(pOrigin,209.77,108.44,6.00),vTravel,z5,tPen\WObj:=wPaper;
    MoveL Offs(pOrigin,209.77,108.44,0.00),v60,z0,tPen\WObj:=wPaper;
    MoveL Offs(pOrigin,209.77,108.92,0.00),v40,z0,tPen\WObj:=wPaper;
    MoveL Offs(pOrigin,210.25,109.39,0.00),v40,z0,tPen\WObj:=wPaper;
    MoveL Offs(pOrigin,209.77,108.44,0.00),v40,z0,tPen\WObj:=wPaper;
    MoveL Offs(pOrigin,209.77,108.92,0.00),v40,z0,tPen\WObj:=wPaper;
    MoveL Offs(pOrigin,210.25,109.39,0.00),v40,z0,tPen\WObj:=wPaper;
    MoveL Offs(pOrigin,209.77,108.44,0.00),v40,fine,tPen\WObj:=wPaper;
    MoveL Offs(pOrigin,209.77,108.44,6.00),v60,z5,tPen\WObj:=wPaper;
    MoveL Offs(pOrigin,210.73,109.87,6.00),vTravel,z5,tPen\WObj:=wPaper;
    MoveL Offs(pOrigin,210.73,109.87,0.00),v60,z0,tPen\WObj:=wPaper;
    MoveL Offs(pOrigin,210.73,110.35,0.00),v40,z0,tPen\WObj:=wPaper;
    MoveL Offs(pOrigin,211.21,110.35,0.00),v40,z0,tPen\WObj:=wPaper;
    MoveL Offs(pOrigin,210.73,109.87,0.00),v40,z0,tPen\WObj:=wPaper;
    MoveL Offs(pOrigin,210.73,110.35,0.00),v40,z0,tPen\WObj:=wPaper;
    MoveL Offs(pOrigin,211.21,110.35,0.00),v40,z0,tPen\WObj:=wPaper;
    MoveL Offs(pOrigin,210.73,109.87,0.00),v40,fine,tPen\WObj:=wPaper;
    MoveL Offs(pOrigin,210.73,109.87,6.00),v60,z5,tPen\WObj:=wPaper;
    MoveL Offs(pOrigin,221.75,86.41,6.00),vTravel,z5,tPen\WObj:=wPaper;
    MoveL Offs(pOrigin,221.75,86.41,0.00),v60,z0,tPen\WObj:=wPaper;
    MoveL Offs(pOrigin,219.35,84.81,0.00),v40,z0,tPen\WObj:=wPaper;
    MoveL Offs(pOrigin,216.48,83.54,0.00),v40,z0,tPen\WObj:=wPaper;
    MoveL Offs(pOrigin,216.16,82.58,0.00),v40,z0,tPen\WObj:=wPaper;
    MoveL Offs(pOrigin,216.96,81.78,0.00),v40,z0,tPen\WObj:=wPaper;
    MoveL Offs(pOrigin,224.14,79.70,0.00),v40,z0,tPen\WObj:=wPaper;
    MoveL Offs(pOrigin,227.49,79.23,0.00),v40,z0,tPen\WObj:=wPaper;
    MoveL Offs(pOrigin,230.85,78.27,0.00),v40,z0,tPen\WObj:=wPaper;
    MoveL Offs(pOrigin,233.72,78.27,0.00),v40,z0,tPen\WObj:=wPaper;
    MoveL Offs(pOrigin,237.55,77.31,0.00),v40,z0,tPen\WObj:=wPaper;
    MoveL Offs(pOrigin,254.79,77.31,0.00),v40,z0,tPen\WObj:=wPaper;
    MoveL Offs(pOrigin,259.10,78.27,0.00),v40,z0,tPen\WObj:=wPaper;
    MoveL Offs(pOrigin,261.01,78.27,0.00),v40,z0,tPen\WObj:=wPaper;
    MoveL Offs(pOrigin,264.37,79.23,0.00),v40,z0,tPen\WObj:=wPaper;
    MoveL Offs(pOrigin,265.80,79.23,0.00),v40,z0,tPen\WObj:=wPaper;
    MoveL Offs(pOrigin,271.07,80.66,0.00),v40,z0,tPen\WObj:=wPaper;
    MoveL Offs(pOrigin,272.51,80.66,0.00),v40,z0,tPen\WObj:=wPaper;
    MoveL Offs(pOrigin,283.52,84.33,0.00),v40,z0,tPen\WObj:=wPaper;
    MoveL Offs(pOrigin,295.97,90.40,0.00),v40,z0,tPen\WObj:=wPaper;
    MoveL Offs(pOrigin,309.86,99.82,0.00),v40,z0,tPen\WObj:=wPaper;
    MoveL Offs(pOrigin,310.82,100.77,0.00),v40,z0,tPen\WObj:=wPaper;
    MoveL Offs(pOrigin,309.86,100.30,0.00),v40,z0,tPen\WObj:=wPaper;
    MoveL Offs(pOrigin,310.82,101.25,0.00),v40,z0,tPen\WObj:=wPaper;
    MoveL Offs(pOrigin,312.25,102.21,0.00),v40,z0,tPen\WObj:=wPaper;
    MoveL Offs(pOrigin,314.65,104.61,0.00),v40,z0,tPen\WObj:=wPaper;
    MoveL Offs(pOrigin,315.13,106.04,0.00),v40,z0,tPen\WObj:=wPaper;
    MoveL Offs(pOrigin,314.65,106.84,0.00),v40,z0,tPen\WObj:=wPaper;
    MoveL Offs(pOrigin,313.69,107.00,0.00),v40,z0,tPen\WObj:=wPaper;
    MoveL Offs(pOrigin,311.77,106.04,0.00),v40,z0,tPen\WObj:=wPaper;
    MoveL Offs(pOrigin,310.82,106.04,0.00),v40,z0,tPen\WObj:=wPaper;
    MoveL Offs(pOrigin,308.42,105.24,0.00),v40,z0,tPen\WObj:=wPaper;
    MoveL Offs(pOrigin,298.37,98.22,0.00),v40,z0,tPen\WObj:=wPaper;
    MoveL Offs(pOrigin,291.18,94.23,0.00),v40,z0,tPen\WObj:=wPaper;
    MoveL Offs(pOrigin,280.17,89.44,0.00),v40,z0,tPen\WObj:=wPaper;
    MoveL Offs(pOrigin,266.76,85.45,0.00),v40,z0,tPen\WObj:=wPaper;
    MoveL Offs(pOrigin,265.32,85.45,0.00),v40,z0,tPen\WObj:=wPaper;
    MoveL Offs(pOrigin,259.58,84.01,0.00),v40,z0,tPen\WObj:=wPaper;
    MoveL Offs(pOrigin,257.18,84.01,0.00),v40,z0,tPen\WObj:=wPaper;
    MoveL Offs(pOrigin,252.87,83.06,0.00),v40,z0,tPen\WObj:=wPaper;
    MoveL Offs(pOrigin,237.07,83.06,0.00),v40,z0,tPen\WObj:=wPaper;
    MoveL Offs(pOrigin,233.24,84.01,0.00),v40,z0,tPen\WObj:=wPaper;
    MoveL Offs(pOrigin,231.80,84.01,0.00),v40,z0,tPen\WObj:=wPaper;
    MoveL Offs(pOrigin,223.18,86.41,0.00),v40,z0,tPen\WObj:=wPaper;
    MoveL Offs(pOrigin,221.75,86.41,0.00),v40,fine,tPen\WObj:=wPaper;
    MoveL Offs(pOrigin,221.75,86.41,6.00),v60,z5,tPen\WObj:=wPaper;
    MoveL Offs(pOrigin,219.83,85.45,6.00),vTravel,z5,tPen\WObj:=wPaper;
    MoveL Offs(pOrigin,219.83,85.45,0.00),v60,z0,tPen\WObj:=wPaper;
    MoveL Offs(pOrigin,220.79,86.41,0.00),v40,z0,tPen\WObj:=wPaper;
    MoveL Offs(pOrigin,219.83,85.45,0.00),v40,fine,tPen\WObj:=wPaper;
    MoveL Offs(pOrigin,219.83,85.45,6.00),v60,z5,tPen\WObj:=wPaper;
    MoveL Offs(pOrigin,210.25,46.66,6.00),vTravel,z5,tPen\WObj:=wPaper;
    MoveL Offs(pOrigin,210.25,46.66,0.00),v60,z0,tPen\WObj:=wPaper;
    MoveL Offs(pOrigin,206.42,46.66,0.00),v40,z0,tPen\WObj:=wPaper;
    MoveL Offs(pOrigin,204.03,45.70,0.00),v40,z0,tPen\WObj:=wPaper;
    MoveL Offs(pOrigin,201.31,42.83,0.00),v40,z0,tPen\WObj:=wPaper;
    MoveL Offs(pOrigin,201.15,39.96,0.00),v40,z0,tPen\WObj:=wPaper;
    MoveL Offs(pOrigin,202.11,38.04,0.00),v40,z0,tPen\WObj:=wPaper;
    MoveL Offs(pOrigin,203.07,37.08,0.00),v40,z0,tPen\WObj:=wPaper;
    MoveL Offs(pOrigin,205.94,35.49,0.00),v40,z0,tPen\WObj:=wPaper;
    MoveL Offs(pOrigin,210.73,34.05,0.00),v40,z0,tPen\WObj:=wPaper;
    MoveL Offs(pOrigin,211.69,32.77,0.00),v40,z0,tPen\WObj:=wPaper;
    MoveL Offs(pOrigin,211.53,31.34,0.00),v40,z0,tPen\WObj:=wPaper;
    MoveL Offs(pOrigin,210.25,30.22,0.00),v40,z0,tPen\WObj:=wPaper;
    MoveL Offs(pOrigin,209.30,29.90,0.00),v40,z0,tPen\WObj:=wPaper;
    MoveL Offs(pOrigin,207.38,29.90,0.00),v40,z0,tPen\WObj:=wPaper;
    MoveL Offs(pOrigin,204.99,30.54,0.00),v40,z0,tPen\WObj:=wPaper;
    MoveL Offs(pOrigin,204.67,31.02,0.00),v40,z0,tPen\WObj:=wPaper;
    MoveL Offs(pOrigin,211.37,40.28,0.00),v40,z0,tPen\WObj:=wPaper;
    MoveL Offs(pOrigin,214.40,45.07,0.00),v40,z0,tPen\WObj:=wPaper;
    MoveL Offs(pOrigin,212.65,46.02,0.00),v40,z0,tPen\WObj:=wPaper;
    MoveL Offs(pOrigin,210.25,46.66,0.00),v40,fine,tPen\WObj:=wPaper;
    MoveL Offs(pOrigin,210.25,46.66,6.00),v60,z5,tPen\WObj:=wPaper;
    MoveL Offs(pOrigin,210.25,43.31,6.00),vTravel,z5,tPen\WObj:=wPaper;
    MoveL Offs(pOrigin,210.25,43.31,0.00),v60,z0,tPen\WObj:=wPaper;
    MoveL Offs(pOrigin,213.13,42.35,0.00),v40,z0,tPen\WObj:=wPaper;
  ENDPROC

  PROC DrawPart8()
    MoveL Offs(pOrigin,214.08,42.83,0.00),v40,z0,tPen\WObj:=wPaper;
    MoveL Offs(pOrigin,214.56,43.79,0.00),v40,z0,tPen\WObj:=wPaper;
    MoveL Offs(pOrigin,210.25,43.31,0.00),v40,z0,tPen\WObj:=wPaper;
    MoveL Offs(pOrigin,209.30,43.31,0.00),v40,z0,tPen\WObj:=wPaper;
    MoveL Offs(pOrigin,204.99,41.87,0.00),v40,z0,tPen\WObj:=wPaper;
    MoveL Offs(pOrigin,204.99,42.35,0.00),v40,z0,tPen\WObj:=wPaper;
    MoveL Offs(pOrigin,205.46,42.83,0.00),v40,z0,tPen\WObj:=wPaper;
    MoveL Offs(pOrigin,205.94,42.83,0.00),v40,z0,tPen\WObj:=wPaper;
    MoveL Offs(pOrigin,206.42,43.31,0.00),v40,z0,tPen\WObj:=wPaper;
    MoveL Offs(pOrigin,209.30,43.31,0.00),v40,z0,tPen\WObj:=wPaper;
    MoveL Offs(pOrigin,204.99,41.87,0.00),v40,z0,tPen\WObj:=wPaper;
    MoveL Offs(pOrigin,204.99,42.35,0.00),v40,z0,tPen\WObj:=wPaper;
    MoveL Offs(pOrigin,205.46,42.83,0.00),v40,z0,tPen\WObj:=wPaper;
    MoveL Offs(pOrigin,205.94,42.83,0.00),v40,z0,tPen\WObj:=wPaper;
    MoveL Offs(pOrigin,206.42,43.31,0.00),v40,z0,tPen\WObj:=wPaper;
    MoveL Offs(pOrigin,209.30,43.31,0.00),v40,fine,tPen\WObj:=wPaper;
    MoveL Offs(pOrigin,209.30,43.31,6.00),v60,z5,tPen\WObj:=wPaper;
    MoveL Offs(pOrigin,206.90,39.48,6.00),vTravel,z5,tPen\WObj:=wPaper;
    MoveL Offs(pOrigin,206.90,39.48,0.00),v60,z0,tPen\WObj:=wPaper;
    MoveL Offs(pOrigin,206.42,39.48,0.00),v40,z0,tPen\WObj:=wPaper;
    MoveL Offs(pOrigin,206.90,39.00,0.00),v40,z0,tPen\WObj:=wPaper;
    MoveL Offs(pOrigin,206.90,39.48,0.00),v40,z0,tPen\WObj:=wPaper;
    MoveL Offs(pOrigin,206.42,39.48,0.00),v40,z0,tPen\WObj:=wPaper;
    MoveL Offs(pOrigin,206.90,39.00,0.00),v40,z0,tPen\WObj:=wPaper;
    MoveL Offs(pOrigin,206.90,39.48,0.00),v40,z0,tPen\WObj:=wPaper;
    MoveL Offs(pOrigin,207.38,39.16,0.00),v40,z0,tPen\WObj:=wPaper;
    MoveL Offs(pOrigin,213.13,37.24,0.00),v40,z0,tPen\WObj:=wPaper;
    MoveL Offs(pOrigin,214.56,36.13,0.00),v40,z0,tPen\WObj:=wPaper;
    MoveL Offs(pOrigin,216.00,33.25,0.00),v40,z0,tPen\WObj:=wPaper;
    MoveL Offs(pOrigin,216.00,31.82,0.00),v40,z0,tPen\WObj:=wPaper;
    MoveL Offs(pOrigin,214.56,28.46,0.00),v40,z0,tPen\WObj:=wPaper;
    MoveL Offs(pOrigin,212.65,27.19,0.00),v40,z0,tPen\WObj:=wPaper;
    MoveL Offs(pOrigin,210.25,26.55,0.00),v40,z0,tPen\WObj:=wPaper;
    MoveL Offs(pOrigin,205.94,26.55,0.00),v40,z0,tPen\WObj:=wPaper;
    MoveL Offs(pOrigin,203.07,27.35,0.00),v40,z0,tPen\WObj:=wPaper;
    MoveL Offs(pOrigin,201.63,28.15,0.00),v40,z0,tPen\WObj:=wPaper;
    MoveL Offs(pOrigin,201.00,28.94,0.00),v40,z0,tPen\WObj:=wPaper;
    MoveL Offs(pOrigin,200.84,29.90,0.00),v40,z0,tPen\WObj:=wPaper;
    MoveL Offs(pOrigin,201.63,31.18,0.00),v40,z0,tPen\WObj:=wPaper;
    MoveL Offs(pOrigin,202.59,31.66,0.00),v40,z0,tPen\WObj:=wPaper;
    MoveL Offs(pOrigin,203.55,31.50,0.00),v40,z0,tPen\WObj:=wPaper;
    MoveL Offs(pOrigin,205.94,40.12,0.00),v40,z0,tPen\WObj:=wPaper;
    MoveL Offs(pOrigin,207.38,39.16,0.00),v40,fine,tPen\WObj:=wPaper;
    MoveL Offs(pOrigin,207.38,39.16,6.00),v60,z5,tPen\WObj:=wPaper;
    MoveL Offs(pOrigin,205.46,39.96,6.00),vTravel,z5,tPen\WObj:=wPaper;
    MoveL Offs(pOrigin,205.46,39.96,0.00),v60,z0,tPen\WObj:=wPaper;
    MoveL Offs(pOrigin,204.99,41.39,0.00),v40,z0,tPen\WObj:=wPaper;
    MoveL Offs(pOrigin,205.46,39.96,0.00),v40,fine,tPen\WObj:=wPaper;
    MoveL Offs(pOrigin,205.46,39.96,6.00),v60,z5,tPen\WObj:=wPaper;
    MoveL Offs(pOrigin,202.11,38.04,6.00),vTravel,z5,tPen\WObj:=wPaper;
    MoveL Offs(pOrigin,202.11,38.04,0.00),v60,z0,tPen\WObj:=wPaper;
    MoveL Offs(pOrigin,201.63,38.04,0.00),v40,z0,tPen\WObj:=wPaper;
    MoveL Offs(pOrigin,202.11,37.56,0.00),v40,z0,tPen\WObj:=wPaper;
    MoveL Offs(pOrigin,202.11,38.04,0.00),v40,z0,tPen\WObj:=wPaper;
    MoveL Offs(pOrigin,201.63,38.04,0.00),v40,z0,tPen\WObj:=wPaper;
    MoveL Offs(pOrigin,202.11,37.56,0.00),v40,z0,tPen\WObj:=wPaper;
    MoveL Offs(pOrigin,202.11,38.04,0.00),v40,fine,tPen\WObj:=wPaper;
    MoveL Offs(pOrigin,202.11,38.04,6.00),v60,z5,tPen\WObj:=wPaper;
    MoveL Offs(pOrigin,201.63,43.79,6.00),vTravel,z5,tPen\WObj:=wPaper;
    MoveL Offs(pOrigin,201.63,43.79,0.00),v60,z0,tPen\WObj:=wPaper;
    MoveL Offs(pOrigin,203.55,45.70,0.00),v40,z0,tPen\WObj:=wPaper;
    MoveL Offs(pOrigin,201.63,43.79,0.00),v40,fine,tPen\WObj:=wPaper;
    MoveL Offs(pOrigin,201.63,43.79,6.00),v60,z5,tPen\WObj:=wPaper;
    MoveL Offs(pOrigin,192.54,41.39,6.00),vTravel,z5,tPen\WObj:=wPaper;
    MoveL Offs(pOrigin,192.54,41.39,0.00),v60,z0,tPen\WObj:=wPaper;
    MoveL Offs(pOrigin,192.06,41.87,0.00),v40,z0,tPen\WObj:=wPaper;
    MoveL Offs(pOrigin,192.54,40.92,0.00),v40,z0,tPen\WObj:=wPaper;
    MoveL Offs(pOrigin,192.54,41.39,0.00),v40,z0,tPen\WObj:=wPaper;
    MoveL Offs(pOrigin,192.06,41.87,0.00),v40,z0,tPen\WObj:=wPaper;
    MoveL Offs(pOrigin,192.54,40.92,0.00),v40,z0,tPen\WObj:=wPaper;
    MoveL Offs(pOrigin,192.54,41.39,0.00),v40,fine,tPen\WObj:=wPaper;
    MoveL Offs(pOrigin,192.54,41.39,6.00),v60,z5,tPen\WObj:=wPaper;
    MoveL Offs(pOrigin,191.90,42.83,6.00),vTravel,z5,tPen\WObj:=wPaper;
    MoveL Offs(pOrigin,191.90,42.83,0.00),v60,z0,tPen\WObj:=wPaper;
    MoveL Offs(pOrigin,189.66,44.91,0.00),v40,z0,tPen\WObj:=wPaper;
    MoveL Offs(pOrigin,187.75,46.02,0.00),v40,z0,tPen\WObj:=wPaper;
    MoveL Offs(pOrigin,185.35,46.66,0.00),v40,z0,tPen\WObj:=wPaper;
    MoveL Offs(pOrigin,182.00,46.66,0.00),v40,z0,tPen\WObj:=wPaper;
    MoveL Offs(pOrigin,179.61,45.86,0.00),v40,z0,tPen\WObj:=wPaper;
    MoveL Offs(pOrigin,177.21,44.27,0.00),v40,z0,tPen\WObj:=wPaper;
    MoveL Offs(pOrigin,174.66,40.92,0.00),v40,z0,tPen\WObj:=wPaper;
    MoveL Offs(pOrigin,173.86,39.00,0.00),v40,z0,tPen\WObj:=wPaper;
    MoveL Offs(pOrigin,173.86,34.21,0.00),v40,z0,tPen\WObj:=wPaper;
    MoveL Offs(pOrigin,174.66,32.30,0.00),v40,z0,tPen\WObj:=wPaper;
    MoveL Offs(pOrigin,176.25,29.90,0.00),v40,z0,tPen\WObj:=wPaper;
    MoveL Offs(pOrigin,177.69,28.46,0.00),v40,z0,tPen\WObj:=wPaper;
    MoveL Offs(pOrigin,179.61,27.19,0.00),v40,z0,tPen\WObj:=wPaper;
    MoveL Offs(pOrigin,181.52,26.55,0.00),v40,z0,tPen\WObj:=wPaper;
    MoveL Offs(pOrigin,186.31,26.55,0.00),v40,z0,tPen\WObj:=wPaper;
    MoveL Offs(pOrigin,188.23,27.35,0.00),v40,z0,tPen\WObj:=wPaper;
    MoveL Offs(pOrigin,190.94,29.10,0.00),v40,z0,tPen\WObj:=wPaper;
    MoveL Offs(pOrigin,191.10,28.94,0.00),v40,z0,tPen\WObj:=wPaper;
    MoveL Offs(pOrigin,192.69,31.82,0.00),v40,z0,tPen\WObj:=wPaper;
    MoveL Offs(pOrigin,193.97,36.13,0.00),v40,z0,tPen\WObj:=wPaper;
    MoveL Offs(pOrigin,193.49,39.00,0.00),v40,z0,tPen\WObj:=wPaper;
    MoveL Offs(pOrigin,191.90,42.83,0.00),v40,z0,tPen\WObj:=wPaper;
    MoveL Offs(pOrigin,191.58,42.83,0.00),v40,z0,tPen\WObj:=wPaper;
    MoveL Offs(pOrigin,191.10,43.79,0.00),v40,z0,tPen\WObj:=wPaper;
    MoveL Offs(pOrigin,191.58,43.31,0.00),v40,z0,tPen\WObj:=wPaper;
    MoveL Offs(pOrigin,191.58,42.83,0.00),v40,z0,tPen\WObj:=wPaper;
    MoveL Offs(pOrigin,191.10,43.79,0.00),v40,z0,tPen\WObj:=wPaper;
    MoveL Offs(pOrigin,191.58,43.31,0.00),v40,z0,tPen\WObj:=wPaper;
    MoveL Offs(pOrigin,191.58,42.83,0.00),v40,fine,tPen\WObj:=wPaper;
    MoveL Offs(pOrigin,191.58,42.83,6.00),v60,z5,tPen\WObj:=wPaper;
    MoveL Offs(pOrigin,190.14,44.27,6.00),vTravel,z5,tPen\WObj:=wPaper;
    MoveL Offs(pOrigin,190.14,44.27,0.00),v60,z0,tPen\WObj:=wPaper;
    MoveL Offs(pOrigin,189.66,45.23,0.00),v40,z0,tPen\WObj:=wPaper;
    MoveL Offs(pOrigin,190.14,44.75,0.00),v40,z0,tPen\WObj:=wPaper;
    MoveL Offs(pOrigin,190.14,44.27,0.00),v40,z0,tPen\WObj:=wPaper;
    MoveL Offs(pOrigin,189.66,45.23,0.00),v40,z0,tPen\WObj:=wPaper;
    MoveL Offs(pOrigin,190.14,44.75,0.00),v40,z0,tPen\WObj:=wPaper;
    MoveL Offs(pOrigin,190.14,44.27,0.00),v40,fine,tPen\WObj:=wPaper;
    MoveL Offs(pOrigin,190.14,44.27,6.00),v60,z5,tPen\WObj:=wPaper;
    MoveL Offs(pOrigin,187.75,42.03,6.00),vTravel,z5,tPen\WObj:=wPaper;
    MoveL Offs(pOrigin,187.75,42.03,0.00),v60,z0,tPen\WObj:=wPaper;
    MoveL Offs(pOrigin,189.34,39.96,0.00),v40,z0,tPen\WObj:=wPaper;
    MoveL Offs(pOrigin,189.66,39.00,0.00),v40,z0,tPen\WObj:=wPaper;
    MoveL Offs(pOrigin,189.66,34.21,0.00),v40,z0,tPen\WObj:=wPaper;
    MoveL Offs(pOrigin,188.70,32.30,0.00),v40,z0,tPen\WObj:=wPaper;
    MoveL Offs(pOrigin,186.79,30.54,0.00),v40,z0,tPen\WObj:=wPaper;
  ENDPROC

  PROC DrawPart9()
    MoveL Offs(pOrigin,184.87,29.90,0.00),v40,z0,tPen\WObj:=wPaper;
    MoveL Offs(pOrigin,183.44,29.90,0.00),v40,z0,tPen\WObj:=wPaper;
    MoveL Offs(pOrigin,181.04,30.54,0.00),v40,z0,tPen\WObj:=wPaper;
    MoveL Offs(pOrigin,178.33,33.73,0.00),v40,z0,tPen\WObj:=wPaper;
    MoveL Offs(pOrigin,177.69,35.65,0.00),v40,z0,tPen\WObj:=wPaper;
    MoveL Offs(pOrigin,177.69,38.04,0.00),v40,z0,tPen\WObj:=wPaper;
    MoveL Offs(pOrigin,178.65,40.44,0.00),v40,z0,tPen\WObj:=wPaper;
    MoveL Offs(pOrigin,181.04,42.67,0.00),v40,z0,tPen\WObj:=wPaper;
    MoveL Offs(pOrigin,182.96,43.31,0.00),v40,z0,tPen\WObj:=wPaper;
    MoveL Offs(pOrigin,185.35,43.31,0.00),v40,z0,tPen\WObj:=wPaper;
    MoveL Offs(pOrigin,187.75,42.03,0.00),v40,fine,tPen\WObj:=wPaper;
    MoveL Offs(pOrigin,187.75,42.03,6.00),v60,z5,tPen\WObj:=wPaper;
    MoveL Offs(pOrigin,181.04,42.35,6.00),vTravel,z5,tPen\WObj:=wPaper;
    MoveL Offs(pOrigin,181.04,42.35,0.00),v60,z0,tPen\WObj:=wPaper;
    MoveL Offs(pOrigin,178.65,39.96,0.00),v40,z0,tPen\WObj:=wPaper;
    MoveL Offs(pOrigin,178.65,40.44,0.00),v40,z0,tPen\WObj:=wPaper;
    MoveL Offs(pOrigin,179.13,40.44,0.00),v40,z0,tPen\WObj:=wPaper;
    MoveL Offs(pOrigin,181.04,42.35,0.00),v40,z0,tPen\WObj:=wPaper;
    MoveL Offs(pOrigin,178.65,39.96,0.00),v40,z0,tPen\WObj:=wPaper;
    MoveL Offs(pOrigin,178.65,40.44,0.00),v40,z0,tPen\WObj:=wPaper;
    MoveL Offs(pOrigin,179.13,40.44,0.00),v40,z0,tPen\WObj:=wPaper;
    MoveL Offs(pOrigin,181.04,42.35,0.00),v40,fine,tPen\WObj:=wPaper;
    MoveL Offs(pOrigin,181.04,42.35,6.00),v60,z5,tPen\WObj:=wPaper;
    MoveL Offs(pOrigin,176.25,43.79,6.00),vTravel,z5,tPen\WObj:=wPaper;
    MoveL Offs(pOrigin,176.25,43.79,0.00),v60,z0,tPen\WObj:=wPaper;
    MoveL Offs(pOrigin,177.21,44.75,0.00),v40,z0,tPen\WObj:=wPaper;
    MoveL Offs(pOrigin,176.25,43.79,0.00),v40,fine,tPen\WObj:=wPaper;
    MoveL Offs(pOrigin,176.25,43.79,6.00),v60,z5,tPen\WObj:=wPaper;
    MoveL Offs(pOrigin,165.24,44.27,6.00),vTravel,z5,tPen\WObj:=wPaper;
    MoveL Offs(pOrigin,165.24,44.27,0.00),v60,z0,tPen\WObj:=wPaper;
    MoveL Offs(pOrigin,164.60,46.02,0.00),v40,z0,tPen\WObj:=wPaper;
    MoveL Offs(pOrigin,162.37,46.02,0.00),v40,z0,tPen\WObj:=wPaper;
    MoveL Offs(pOrigin,161.41,44.75,0.00),v40,z0,tPen\WObj:=wPaper;
    MoveL Offs(pOrigin,161.41,32.30,0.00),v40,z0,tPen\WObj:=wPaper;
    MoveL Offs(pOrigin,161.09,31.34,0.00),v40,z0,tPen\WObj:=wPaper;
    MoveL Offs(pOrigin,160.45,30.54,0.00),v40,z0,tPen\WObj:=wPaper;
    MoveL Offs(pOrigin,158.54,29.90,0.00),v40,z0,tPen\WObj:=wPaper;
    MoveL Offs(pOrigin,155.66,30.54,0.00),v40,z0,tPen\WObj:=wPaper;
    MoveL Offs(pOrigin,154.70,30.38,0.00),v40,z0,tPen\WObj:=wPaper;
    MoveL Offs(pOrigin,153.43,28.94,0.00),v40,z0,tPen\WObj:=wPaper;
    MoveL Offs(pOrigin,153.75,27.99,0.00),v40,z0,tPen\WObj:=wPaper;
    MoveL Offs(pOrigin,154.70,27.19,0.00),v40,z0,tPen\WObj:=wPaper;
    MoveL Offs(pOrigin,156.62,26.55,0.00),v40,z0,tPen\WObj:=wPaper;
    MoveL Offs(pOrigin,159.97,26.55,0.00),v40,z0,tPen\WObj:=wPaper;
    MoveL Offs(pOrigin,162.85,27.99,0.00),v40,z0,tPen\WObj:=wPaper;
    MoveL Offs(pOrigin,164.60,30.38,0.00),v40,z0,tPen\WObj:=wPaper;
    MoveL Offs(pOrigin,165.24,32.30,0.00),v40,z0,tPen\WObj:=wPaper;
    MoveL Offs(pOrigin,165.24,39.48,0.00),v40,z0,tPen\WObj:=wPaper;
    MoveL Offs(pOrigin,164.76,40.92,0.00),v40,z0,tPen\WObj:=wPaper;
    MoveL Offs(pOrigin,165.24,44.27,0.00),v40,fine,tPen\WObj:=wPaper;
    MoveL Offs(pOrigin,165.24,44.27,6.00),v60,z5,tPen\WObj:=wPaper;
    MoveL Offs(pOrigin,174.34,32.30,6.00),vTravel,z5,tPen\WObj:=wPaper;
    MoveL Offs(pOrigin,174.34,32.30,0.00),v60,z0,tPen\WObj:=wPaper;
    MoveL Offs(pOrigin,174.82,31.34,0.00),v40,z0,tPen\WObj:=wPaper;
    MoveL Offs(pOrigin,174.82,31.82,0.00),v40,z0,tPen\WObj:=wPaper;
    MoveL Offs(pOrigin,174.34,32.30,0.00),v40,z0,tPen\WObj:=wPaper;
    MoveL Offs(pOrigin,174.82,31.34,0.00),v40,z0,tPen\WObj:=wPaper;
    MoveL Offs(pOrigin,174.82,31.82,0.00),v40,z0,tPen\WObj:=wPaper;
    MoveL Offs(pOrigin,174.34,32.30,0.00),v40,fine,tPen\WObj:=wPaper;
    MoveL Offs(pOrigin,174.34,32.30,6.00),v60,z5,tPen\WObj:=wPaper;
    MoveL Offs(pOrigin,175.77,29.90,6.00),vTravel,z5,tPen\WObj:=wPaper;
    MoveL Offs(pOrigin,175.77,29.90,0.00),v60,z0,tPen\WObj:=wPaper;
    MoveL Offs(pOrigin,176.73,28.94,0.00),v40,z0,tPen\WObj:=wPaper;
    MoveL Offs(pOrigin,176.73,29.42,0.00),v40,z0,tPen\WObj:=wPaper;
    MoveL Offs(pOrigin,176.25,29.42,0.00),v40,z0,tPen\WObj:=wPaper;
    MoveL Offs(pOrigin,175.77,29.90,0.00),v40,z0,tPen\WObj:=wPaper;
    MoveL Offs(pOrigin,176.73,28.94,0.00),v40,z0,tPen\WObj:=wPaper;
    MoveL Offs(pOrigin,176.73,29.42,0.00),v40,z0,tPen\WObj:=wPaper;
    MoveL Offs(pOrigin,176.25,29.42,0.00),v40,z0,tPen\WObj:=wPaper;
    MoveL Offs(pOrigin,175.77,29.90,0.00),v40,fine,tPen\WObj:=wPaper;
    MoveL Offs(pOrigin,175.77,29.90,6.00),v60,z5,tPen\WObj:=wPaper;
    MoveL Offs(pOrigin,179.61,32.30,6.00),vTravel,z5,tPen\WObj:=wPaper;
    MoveL Offs(pOrigin,179.61,32.30,0.00),v60,z0,tPen\WObj:=wPaper;
    MoveL Offs(pOrigin,180.08,31.34,0.00),v40,z0,tPen\WObj:=wPaper;
    MoveL Offs(pOrigin,180.08,31.82,0.00),v40,z0,tPen\WObj:=wPaper;
    MoveL Offs(pOrigin,179.61,32.30,0.00),v40,z0,tPen\WObj:=wPaper;
    MoveL Offs(pOrigin,180.08,31.34,0.00),v40,z0,tPen\WObj:=wPaper;
    MoveL Offs(pOrigin,180.08,31.82,0.00),v40,z0,tPen\WObj:=wPaper;
    MoveL Offs(pOrigin,179.61,32.30,0.00),v40,fine,tPen\WObj:=wPaper;
    MoveL Offs(pOrigin,179.61,32.30,6.00),v60,z5,tPen\WObj:=wPaper;
    MoveL Offs(pOrigin,186.79,30.86,6.00),vTravel,z5,tPen\WObj:=wPaper;
    MoveL Offs(pOrigin,186.79,30.86,0.00),v60,z0,tPen\WObj:=wPaper;
    MoveL Offs(pOrigin,187.75,31.82,0.00),v40,z0,tPen\WObj:=wPaper;
    MoveL Offs(pOrigin,186.79,30.86,0.00),v40,fine,tPen\WObj:=wPaper;
    MoveL Offs(pOrigin,186.79,30.86,6.00),v60,z5,tPen\WObj:=wPaper;
    MoveL Offs(pOrigin,201.63,28.46,6.00),vTravel,z5,tPen\WObj:=wPaper;
    MoveL Offs(pOrigin,201.63,28.46,0.00),v60,z0,tPen\WObj:=wPaper;
    MoveL Offs(pOrigin,202.11,27.99,0.00),v40,z0,tPen\WObj:=wPaper;
    MoveL Offs(pOrigin,202.59,27.99,0.00),v40,z0,tPen\WObj:=wPaper;
    MoveL Offs(pOrigin,201.63,28.46,0.00),v40,z0,tPen\WObj:=wPaper;
    MoveL Offs(pOrigin,202.11,27.99,0.00),v40,z0,tPen\WObj:=wPaper;
    MoveL Offs(pOrigin,202.59,27.99,0.00),v40,z0,tPen\WObj:=wPaper;
    MoveL Offs(pOrigin,201.63,28.46,0.00),v40,fine,tPen\WObj:=wPaper;
    MoveL Offs(pOrigin,201.63,28.46,6.00),v60,z5,tPen\WObj:=wPaper;
    MoveL Offs(pOrigin,213.13,27.99,6.00),vTravel,z5,tPen\WObj:=wPaper;
    MoveL Offs(pOrigin,213.13,27.99,0.00),v60,z0,tPen\WObj:=wPaper;
    MoveL Offs(pOrigin,213.61,27.99,0.00),v40,z0,tPen\WObj:=wPaper;
    MoveL Offs(pOrigin,214.56,28.94,0.00),v40,z0,tPen\WObj:=wPaper;
    MoveL Offs(pOrigin,213.13,27.99,0.00),v40,z0,tPen\WObj:=wPaper;
    MoveL Offs(pOrigin,213.61,27.99,0.00),v40,z0,tPen\WObj:=wPaper;
    MoveL Offs(pOrigin,214.56,28.94,0.00),v40,z0,tPen\WObj:=wPaper;
    MoveL Offs(pOrigin,213.13,27.99,0.00),v40,fine,tPen\WObj:=wPaper;
    MoveL Offs(pOrigin,213.13,27.99,6.00),v60,z5,tPen\WObj:=wPaper;
    MoveL Offs(pOrigin,215.04,34.69,6.00),vTravel,z5,tPen\WObj:=wPaper;
    MoveL Offs(pOrigin,215.04,34.69,0.00),v60,z0,tPen\WObj:=wPaper;
    MoveL Offs(pOrigin,215.04,35.17,0.00),v40,z0,tPen\WObj:=wPaper;
    MoveL Offs(pOrigin,214.56,35.65,0.00),v40,z0,tPen\WObj:=wPaper;
    MoveL Offs(pOrigin,215.04,34.69,0.00),v40,z0,tPen\WObj:=wPaper;
    MoveL Offs(pOrigin,215.04,35.17,0.00),v40,z0,tPen\WObj:=wPaper;
    MoveL Offs(pOrigin,214.56,35.65,0.00),v40,z0,tPen\WObj:=wPaper;
    MoveL Offs(pOrigin,215.04,34.69,0.00),v40,fine,tPen\WObj:=wPaper;
    MoveL Offs(pOrigin,215.04,34.69,6.00),v60,z5,tPen\WObj:=wPaper;
    MoveL Offs(pOrigin,225.74,31.82,6.00),vTravel,z5,tPen\WObj:=wPaper;
    MoveL Offs(pOrigin,225.74,31.82,0.00),v60,z0,tPen\WObj:=wPaper;
    MoveL Offs(pOrigin,227.49,32.77,0.00),v40,z0,tPen\WObj:=wPaper;
    MoveL Offs(pOrigin,230.37,32.62,0.00),v40,z0,tPen\WObj:=wPaper;
    MoveL Offs(pOrigin,232.12,30.86,0.00),v40,z0,tPen\WObj:=wPaper;
    MoveL Offs(pOrigin,232.12,28.46,0.00),v40,z0,tPen\WObj:=wPaper;
    MoveL Offs(pOrigin,230.37,26.71,0.00),v40,z0,tPen\WObj:=wPaper;
    MoveL Offs(pOrigin,227.17,26.71,0.00),v40,z0,tPen\WObj:=wPaper;
  ENDPROC

  PROC DrawPart10()
    MoveL Offs(pOrigin,225.74,27.99,0.00),v40,z0,tPen\WObj:=wPaper;
    MoveL Offs(pOrigin,225.10,29.42,0.00),v40,z0,tPen\WObj:=wPaper;
    MoveL Offs(pOrigin,225.74,31.82,0.00),v40,fine,tPen\WObj:=wPaper;
    MoveL Offs(pOrigin,225.74,31.82,6.00),v60,z5,tPen\WObj:=wPaper;
    MoveL Offs(pOrigin,226.06,27.99,6.00),vTravel,z5,tPen\WObj:=wPaper;
    MoveL Offs(pOrigin,226.06,27.99,0.00),v60,z0,tPen\WObj:=wPaper;
    MoveL Offs(pOrigin,226.54,27.03,0.00),v40,z0,tPen\WObj:=wPaper;
    MoveL Offs(pOrigin,226.54,27.51,0.00),v40,z0,tPen\WObj:=wPaper;
    MoveL Offs(pOrigin,226.06,27.99,0.00),v40,z0,tPen\WObj:=wPaper;
    MoveL Offs(pOrigin,226.54,27.03,0.00),v40,z0,tPen\WObj:=wPaper;
    MoveL Offs(pOrigin,226.54,27.51,0.00),v40,z0,tPen\WObj:=wPaper;
    MoveL Offs(pOrigin,226.06,27.99,0.00),v40,fine,tPen\WObj:=wPaper;
    MoveL Offs(pOrigin,226.06,27.99,6.00),v60,z5,tPen\WObj:=wPaper;
    MoveL Offs(pOrigin,230.85,27.51,6.00),vTravel,z5,tPen\WObj:=wPaper;
    MoveL Offs(pOrigin,230.85,27.51,0.00),v60,z0,tPen\WObj:=wPaper;
    MoveL Offs(pOrigin,231.80,28.46,0.00),v40,z0,tPen\WObj:=wPaper;
    MoveL Offs(pOrigin,230.85,27.51,0.00),v40,fine,tPen\WObj:=wPaper;
    MoveL Offs(pOrigin,230.85,27.51,6.00),v60,z5,tPen\WObj:=wPaper;
    MoveL Offs(pOrigin,231.80,30.86,6.00),vTravel,z5,tPen\WObj:=wPaper;
    MoveL Offs(pOrigin,231.80,30.86,0.00),v60,z0,tPen\WObj:=wPaper;
    MoveL Offs(pOrigin,231.80,31.34,0.00),v40,z0,tPen\WObj:=wPaper;
    MoveL Offs(pOrigin,231.32,31.34,0.00),v40,z0,tPen\WObj:=wPaper;
    MoveL Offs(pOrigin,230.37,32.30,0.00),v40,z0,tPen\WObj:=wPaper;
    MoveL Offs(pOrigin,231.80,30.86,0.00),v40,z0,tPen\WObj:=wPaper;
    MoveL Offs(pOrigin,231.80,31.34,0.00),v40,z0,tPen\WObj:=wPaper;
    MoveL Offs(pOrigin,231.32,31.34,0.00),v40,z0,tPen\WObj:=wPaper;
    MoveL Offs(pOrigin,230.37,32.30,0.00),v40,z0,tPen\WObj:=wPaper;
    MoveL Offs(pOrigin,231.80,30.86,0.00),v40,fine,tPen\WObj:=wPaper;
    MoveL Offs(pOrigin,231.80,30.86,6.00),v60,z5,tPen\WObj:=wPaper;
    MoveL Offs(pOrigin,242.34,28.94,6.00),vTravel,z5,tPen\WObj:=wPaper;
    MoveL Offs(pOrigin,242.34,28.94,0.00),v60,z0,tPen\WObj:=wPaper;
    MoveL Offs(pOrigin,242.34,33.73,0.00),v40,z0,tPen\WObj:=wPaper;
    MoveL Offs(pOrigin,242.34,28.94,0.00),v40,fine,tPen\WObj:=wPaper;
    MoveL Offs(pOrigin,242.34,28.94,6.00),v60,z5,tPen\WObj:=wPaper;
    MoveL Offs(pOrigin,242.34,27.03,6.00),vTravel,z5,tPen\WObj:=wPaper;
    MoveL Offs(pOrigin,242.34,27.03,0.00),v60,z0,tPen\WObj:=wPaper;
    MoveL Offs(pOrigin,242.34,28.46,0.00),v40,z0,tPen\WObj:=wPaper;
    MoveL Offs(pOrigin,242.34,27.03,0.00),v40,fine,tPen\WObj:=wPaper;
    MoveL Offs(pOrigin,242.34,27.03,6.00),v60,z5,tPen\WObj:=wPaper;
    MoveL Offs(pOrigin,243.77,26.55,6.00),vTravel,z5,tPen\WObj:=wPaper;
    MoveL Offs(pOrigin,243.77,26.55,0.00),v60,z0,tPen\WObj:=wPaper;
    MoveL Offs(pOrigin,244.73,26.55,0.00),v40,z0,tPen\WObj:=wPaper;
    MoveL Offs(pOrigin,245.69,27.51,0.00),v40,z0,tPen\WObj:=wPaper;
    MoveL Offs(pOrigin,245.69,27.03,0.00),v40,z0,tPen\WObj:=wPaper;
    MoveL Offs(pOrigin,243.77,26.55,0.00),v40,z0,tPen\WObj:=wPaper;
    MoveL Offs(pOrigin,244.73,26.55,0.00),v40,z0,tPen\WObj:=wPaper;
    MoveL Offs(pOrigin,245.69,27.51,0.00),v40,z0,tPen\WObj:=wPaper;
    MoveL Offs(pOrigin,245.69,27.03,0.00),v40,z0,tPen\WObj:=wPaper;
    MoveL Offs(pOrigin,243.77,26.55,0.00),v40,fine,tPen\WObj:=wPaper;
    MoveL Offs(pOrigin,243.77,26.55,6.00),v60,z5,tPen\WObj:=wPaper;
    MoveL Offs(pOrigin,245.69,27.99,6.00),vTravel,z5,tPen\WObj:=wPaper;
    MoveL Offs(pOrigin,245.69,27.99,0.00),v60,z0,tPen\WObj:=wPaper;
    MoveL Offs(pOrigin,245.69,29.42,0.00),v40,z0,tPen\WObj:=wPaper;
    MoveL Offs(pOrigin,245.69,27.99,0.00),v40,fine,tPen\WObj:=wPaper;
    MoveL Offs(pOrigin,245.69,27.99,6.00),v60,z5,tPen\WObj:=wPaper;
    MoveL Offs(pOrigin,245.69,30.38,6.00),vTravel,z5,tPen\WObj:=wPaper;
    MoveL Offs(pOrigin,245.69,30.38,0.00),v60,z0,tPen\WObj:=wPaper;
    MoveL Offs(pOrigin,245.69,31.34,0.00),v40,z0,tPen\WObj:=wPaper;
    MoveL Offs(pOrigin,246.65,33.57,0.00),v40,z0,tPen\WObj:=wPaper;
    MoveL Offs(pOrigin,252.87,34.21,0.00),v40,z0,tPen\WObj:=wPaper;
    MoveL Offs(pOrigin,256.07,36.29,0.00),v40,z0,tPen\WObj:=wPaper;
    MoveL Offs(pOrigin,255.75,35.65,0.00),v40,z0,tPen\WObj:=wPaper;
    MoveL Offs(pOrigin,252.23,33.57,0.00),v40,z0,tPen\WObj:=wPaper;
    MoveL Offs(pOrigin,245.69,30.38,0.00),v40,fine,tPen\WObj:=wPaper;
    MoveL Offs(pOrigin,245.69,30.38,6.00),v60,z5,tPen\WObj:=wPaper;
    MoveL Offs(pOrigin,242.34,34.69,6.00),vTravel,z5,tPen\WObj:=wPaper;
    MoveL Offs(pOrigin,242.34,34.69,0.00),v60,z0,tPen\WObj:=wPaper;
    MoveL Offs(pOrigin,242.34,45.70,0.00),v40,z0,tPen\WObj:=wPaper;
    MoveL Offs(pOrigin,242.82,46.18,0.00),v40,z0,tPen\WObj:=wPaper;
    MoveL Offs(pOrigin,247.61,46.66,0.00),v40,z0,tPen\WObj:=wPaper;
    MoveL Offs(pOrigin,244.25,38.52,0.00),v40,z0,tPen\WObj:=wPaper;
    MoveL Offs(pOrigin,242.34,34.69,0.00),v40,fine,tPen\WObj:=wPaper;
    MoveL Offs(pOrigin,242.34,34.69,6.00),v60,z5,tPen\WObj:=wPaper;
    MoveL Offs(pOrigin,246.33,37.56,6.00),vTravel,z5,tPen\WObj:=wPaper;
    MoveL Offs(pOrigin,246.33,37.56,0.00),v60,z0,tPen\WObj:=wPaper;
    MoveL Offs(pOrigin,246.33,43.15,0.00),v40,z0,tPen\WObj:=wPaper;
    MoveL Offs(pOrigin,250.48,43.31,0.00),v40,z0,tPen\WObj:=wPaper;
    MoveL Offs(pOrigin,252.39,42.51,0.00),v40,z0,tPen\WObj:=wPaper;
    MoveL Offs(pOrigin,253.03,41.87,0.00),v40,z0,tPen\WObj:=wPaper;
    MoveL Offs(pOrigin,253.35,39.48,0.00),v40,z0,tPen\WObj:=wPaper;
    MoveL Offs(pOrigin,252.39,37.72,0.00),v40,z0,tPen\WObj:=wPaper;
    MoveL Offs(pOrigin,250.48,37.08,0.00),v40,z0,tPen\WObj:=wPaper;
    MoveL Offs(pOrigin,247.13,37.08,0.00),v40,z0,tPen\WObj:=wPaper;
    MoveL Offs(pOrigin,246.33,37.56,0.00),v40,fine,tPen\WObj:=wPaper;
    MoveL Offs(pOrigin,246.33,37.56,6.00),v60,z5,tPen\WObj:=wPaper;
    MoveL Offs(pOrigin,252.39,38.04,6.00),vTravel,z5,tPen\WObj:=wPaper;
    MoveL Offs(pOrigin,252.39,38.04,0.00),v60,z0,tPen\WObj:=wPaper;
    MoveL Offs(pOrigin,252.87,38.52,0.00),v40,z0,tPen\WObj:=wPaper;
    MoveL Offs(pOrigin,252.87,39.00,0.00),v40,z0,tPen\WObj:=wPaper;
    MoveL Offs(pOrigin,252.39,38.04,0.00),v40,z0,tPen\WObj:=wPaper;
    MoveL Offs(pOrigin,252.87,38.52,0.00),v40,z0,tPen\WObj:=wPaper;
    MoveL Offs(pOrigin,252.87,39.00,0.00),v40,z0,tPen\WObj:=wPaper;
    MoveL Offs(pOrigin,252.39,38.04,0.00),v40,fine,tPen\WObj:=wPaper;
    MoveL Offs(pOrigin,252.39,38.04,6.00),v60,z5,tPen\WObj:=wPaper;
    MoveL Offs(pOrigin,256.70,37.08,6.00),vTravel,z5,tPen\WObj:=wPaper;
    MoveL Offs(pOrigin,256.70,37.08,0.00),v60,z0,tPen\WObj:=wPaper;
    MoveL Offs(pOrigin,257.66,39.48,0.00),v40,z0,tPen\WObj:=wPaper;
    MoveL Offs(pOrigin,257.66,40.44,0.00),v40,z0,tPen\WObj:=wPaper;
    MoveL Offs(pOrigin,256.86,43.31,0.00),v40,z0,tPen\WObj:=wPaper;
    MoveL Offs(pOrigin,255.43,44.91,0.00),v40,z0,tPen\WObj:=wPaper;
    MoveL Offs(pOrigin,256.70,37.08,0.00),v40,fine,tPen\WObj:=wPaper;
    MoveL Offs(pOrigin,256.70,37.08,6.00),v60,z5,tPen\WObj:=wPaper;
    MoveL Offs(pOrigin,254.47,45.38,6.00),vTravel,z5,tPen\WObj:=wPaper;
    MoveL Offs(pOrigin,254.47,45.38,0.00),v60,z0,tPen\WObj:=wPaper;
    MoveL Offs(pOrigin,249.04,46.66,0.00),v40,z0,tPen\WObj:=wPaper;
    MoveL Offs(pOrigin,250.96,46.66,0.00),v40,z0,tPen\WObj:=wPaper;
    MoveL Offs(pOrigin,253.35,46.18,0.00),v40,z0,tPen\WObj:=wPaper;
    MoveL Offs(pOrigin,254.47,45.38,0.00),v40,fine,tPen\WObj:=wPaper;
    MoveL Offs(pOrigin,254.47,45.38,6.00),v60,z5,tPen\WObj:=wPaper;
    MoveL Offs(pOrigin,266.28,45.23,6.00),vTravel,z5,tPen\WObj:=wPaper;
    MoveL Offs(pOrigin,266.28,45.23,0.00),v60,z0,tPen\WObj:=wPaper;
    MoveL Offs(pOrigin,266.76,46.02,0.00),v40,z0,tPen\WObj:=wPaper;
    MoveL Offs(pOrigin,269.15,46.18,0.00),v40,z0,tPen\WObj:=wPaper;
    MoveL Offs(pOrigin,269.95,45.70,0.00),v40,z0,tPen\WObj:=wPaper;
    MoveL Offs(pOrigin,270.11,45.23,0.00),v40,z0,tPen\WObj:=wPaper;
    MoveL Offs(pOrigin,270.11,28.46,0.00),v40,z0,tPen\WObj:=wPaper;
    MoveL Offs(pOrigin,269.15,26.71,0.00),v40,z0,tPen\WObj:=wPaper;
    MoveL Offs(pOrigin,267.72,26.55,0.00),v40,z0,tPen\WObj:=wPaper;
    MoveL Offs(pOrigin,266.76,26.87,0.00),v40,z0,tPen\WObj:=wPaper;
    MoveL Offs(pOrigin,266.28,27.51,0.00),v40,z0,tPen\WObj:=wPaper;
  ENDPROC

  PROC DrawPart11()
    MoveL Offs(pOrigin,266.28,45.23,0.00),v40,fine,tPen\WObj:=wPaper;
    MoveL Offs(pOrigin,266.28,45.23,6.00),v60,z5,tPen\WObj:=wPaper;
    MoveL Offs(pOrigin,280.17,44.75,6.00),vTravel,z5,tPen\WObj:=wPaper;
    MoveL Offs(pOrigin,280.17,44.75,0.00),v60,z0,tPen\WObj:=wPaper;
    MoveL Offs(pOrigin,280.33,44.27,0.00),v40,z0,tPen\WObj:=wPaper;
    MoveL Offs(pOrigin,281.61,43.31,0.00),v40,z0,tPen\WObj:=wPaper;
    MoveL Offs(pOrigin,288.79,43.31,0.00),v40,z0,tPen\WObj:=wPaper;
    MoveL Offs(pOrigin,289.27,42.83,0.00),v40,z0,tPen\WObj:=wPaper;
    MoveL Offs(pOrigin,289.27,41.87,0.00),v40,z0,tPen\WObj:=wPaper;
    MoveL Offs(pOrigin,288.79,40.92,0.00),v40,z0,tPen\WObj:=wPaper;
    MoveL Offs(pOrigin,280.33,29.90,0.00),v40,z0,tPen\WObj:=wPaper;
    MoveL Offs(pOrigin,280.17,27.99,0.00),v40,z0,tPen\WObj:=wPaper;
    MoveL Offs(pOrigin,280.65,27.03,0.00),v40,z0,tPen\WObj:=wPaper;
    MoveL Offs(pOrigin,281.61,26.55,0.00),v40,z0,tPen\WObj:=wPaper;
    MoveL Offs(pOrigin,293.10,26.55,0.00),v40,z0,tPen\WObj:=wPaper;
    MoveL Offs(pOrigin,295.33,27.51,0.00),v40,z0,tPen\WObj:=wPaper;
    MoveL Offs(pOrigin,295.49,28.94,0.00),v40,z0,tPen\WObj:=wPaper;
    MoveL Offs(pOrigin,295.01,29.74,0.00),v40,z0,tPen\WObj:=wPaper;
    MoveL Offs(pOrigin,291.18,29.90,0.00),v40,z0,tPen\WObj:=wPaper;
    MoveL Offs(pOrigin,289.75,30.38,0.00),v40,z0,tPen\WObj:=wPaper;
    MoveL Offs(pOrigin,286.87,30.38,0.00),v40,z0,tPen\WObj:=wPaper;
    MoveL Offs(pOrigin,286.08,30.86,0.00),v40,z0,tPen\WObj:=wPaper;
    MoveL Offs(pOrigin,286.23,31.82,0.00),v40,z0,tPen\WObj:=wPaper;
    MoveL Offs(pOrigin,287.83,34.21,0.00),v40,z0,tPen\WObj:=wPaper;
    MoveL Offs(pOrigin,295.17,43.79,0.00),v40,z0,tPen\WObj:=wPaper;
    MoveL Offs(pOrigin,295.49,45.23,0.00),v40,z0,tPen\WObj:=wPaper;
    MoveL Offs(pOrigin,295.01,46.02,0.00),v40,z0,tPen\WObj:=wPaper;
    MoveL Offs(pOrigin,292.14,46.66,0.00),v40,z0,tPen\WObj:=wPaper;
    MoveL Offs(pOrigin,290.70,46.18,0.00),v40,z0,tPen\WObj:=wPaper;
    MoveL Offs(pOrigin,281.61,46.18,0.00),v40,z0,tPen\WObj:=wPaper;
    MoveL Offs(pOrigin,280.65,45.70,0.00),v40,z0,tPen\WObj:=wPaper;
    MoveL Offs(pOrigin,280.17,44.75,0.00),v40,fine,tPen\WObj:=wPaper;
    MoveL Offs(pOrigin,280.17,44.75,6.00),v60,z5,tPen\WObj:=wPaper;
    MoveL Offs(pOrigin,287.35,39.48,6.00),vTravel,z5,tPen\WObj:=wPaper;
    MoveL Offs(pOrigin,287.35,39.48,0.00),v60,z0,tPen\WObj:=wPaper;
    MoveL Offs(pOrigin,288.79,41.39,0.00),v40,z0,tPen\WObj:=wPaper;
    MoveL Offs(pOrigin,287.35,39.48,0.00),v40,fine,tPen\WObj:=wPaper;
    MoveL Offs(pOrigin,287.35,39.48,6.00),v60,z5,tPen\WObj:=wPaper;
    MoveL Offs(pOrigin,290.70,38.04,6.00),vTravel,z5,tPen\WObj:=wPaper;
    MoveL Offs(pOrigin,290.70,38.04,0.00),v60,z0,tPen\WObj:=wPaper;
    MoveL Offs(pOrigin,291.18,38.04,0.00),v40,z0,tPen\WObj:=wPaper;
    MoveL Offs(pOrigin,291.66,38.52,0.00),v40,z0,tPen\WObj:=wPaper;
    MoveL Offs(pOrigin,290.70,37.56,0.00),v40,z0,tPen\WObj:=wPaper;
    MoveL Offs(pOrigin,290.70,38.04,0.00),v40,z0,tPen\WObj:=wPaper;
    MoveL Offs(pOrigin,291.18,38.04,0.00),v40,z0,tPen\WObj:=wPaper;
    MoveL Offs(pOrigin,291.66,38.52,0.00),v40,z0,tPen\WObj:=wPaper;
    MoveL Offs(pOrigin,290.70,37.56,0.00),v40,z0,tPen\WObj:=wPaper;
    MoveL Offs(pOrigin,290.70,38.04,0.00),v40,fine,tPen\WObj:=wPaper;
    MoveL Offs(pOrigin,290.70,38.04,6.00),v60,z5,tPen\WObj:=wPaper;
    MoveL Offs(pOrigin,290.23,36.61,6.00),vTravel,z5,tPen\WObj:=wPaper;
    MoveL Offs(pOrigin,290.23,36.61,0.00),v60,z0,tPen\WObj:=wPaper;
    MoveL Offs(pOrigin,289.75,36.13,0.00),v40,z0,tPen\WObj:=wPaper;
    MoveL Offs(pOrigin,289.75,36.61,0.00),v40,z0,tPen\WObj:=wPaper;
    MoveL Offs(pOrigin,290.23,36.61,0.00),v40,z0,tPen\WObj:=wPaper;
    MoveL Offs(pOrigin,289.75,36.13,0.00),v40,z0,tPen\WObj:=wPaper;
    MoveL Offs(pOrigin,289.75,36.61,0.00),v40,z0,tPen\WObj:=wPaper;
    MoveL Offs(pOrigin,290.23,36.61,0.00),v40,fine,tPen\WObj:=wPaper;
    MoveL Offs(pOrigin,290.23,36.61,6.00),v60,z5,tPen\WObj:=wPaper;
    MoveL Offs(pOrigin,289.27,35.65,6.00),vTravel,z5,tPen\WObj:=wPaper;
    MoveL Offs(pOrigin,289.27,35.65,0.00),v60,z0,tPen\WObj:=wPaper;
    MoveL Offs(pOrigin,288.79,34.69,0.00),v40,z0,tPen\WObj:=wPaper;
    MoveL Offs(pOrigin,288.79,35.17,0.00),v40,z0,tPen\WObj:=wPaper;
    MoveL Offs(pOrigin,289.27,35.65,0.00),v40,z0,tPen\WObj:=wPaper;
    MoveL Offs(pOrigin,288.79,34.69,0.00),v40,z0,tPen\WObj:=wPaper;
    MoveL Offs(pOrigin,288.79,35.17,0.00),v40,z0,tPen\WObj:=wPaper;
    MoveL Offs(pOrigin,289.27,35.65,0.00),v40,fine,tPen\WObj:=wPaper;
    MoveL Offs(pOrigin,289.27,35.65,6.00),v60,z5,tPen\WObj:=wPaper;
    MoveL Offs(pOrigin,287.35,32.77,6.00),vTravel,z5,tPen\WObj:=wPaper;
    MoveL Offs(pOrigin,287.35,32.77,0.00),v60,z0,tPen\WObj:=wPaper;
    MoveL Offs(pOrigin,286.87,32.30,0.00),v40,z0,tPen\WObj:=wPaper;
    MoveL Offs(pOrigin,286.87,32.77,0.00),v40,z0,tPen\WObj:=wPaper;
    MoveL Offs(pOrigin,287.35,32.77,0.00),v40,z0,tPen\WObj:=wPaper;
    MoveL Offs(pOrigin,286.87,32.30,0.00),v40,z0,tPen\WObj:=wPaper;
    MoveL Offs(pOrigin,286.87,32.77,0.00),v40,z0,tPen\WObj:=wPaper;
    MoveL Offs(pOrigin,287.35,32.77,0.00),v40,fine,tPen\WObj:=wPaper;
    MoveL Offs(pOrigin,287.35,32.77,6.00),v60,z5,tPen\WObj:=wPaper;
    MoveL Offs(pOrigin,284.96,36.61,6.00),vTravel,z5,tPen\WObj:=wPaper;
    MoveL Offs(pOrigin,284.96,36.61,0.00),v60,z0,tPen\WObj:=wPaper;
    MoveL Offs(pOrigin,285.92,37.56,0.00),v40,z0,tPen\WObj:=wPaper;
    MoveL Offs(pOrigin,284.96,36.61,0.00),v40,fine,tPen\WObj:=wPaper;
    MoveL Offs(pOrigin,284.96,36.61,6.00),v60,z5,tPen\WObj:=wPaper;
    MoveL Offs(pOrigin,281.61,32.30,6.00),vTravel,z5,tPen\WObj:=wPaper;
    MoveL Offs(pOrigin,281.61,32.30,0.00),v60,z0,tPen\WObj:=wPaper;
    MoveL Offs(pOrigin,283.04,33.73,0.00),v40,z0,tPen\WObj:=wPaper;
    MoveL Offs(pOrigin,281.61,32.30,0.00),v40,fine,tPen\WObj:=wPaper;
    MoveL Offs(pOrigin,281.61,32.30,6.00),v60,z5,tPen\WObj:=wPaper;
    MoveL Offs(pOrigin,280.17,30.38,6.00),vTravel,z5,tPen\WObj:=wPaper;
    MoveL Offs(pOrigin,280.17,30.38,0.00),v60,z0,tPen\WObj:=wPaper;
    MoveL Offs(pOrigin,281.13,31.34,0.00),v40,z0,tPen\WObj:=wPaper;
    MoveL Offs(pOrigin,280.17,30.38,0.00),v40,fine,tPen\WObj:=wPaper;
    MoveL Offs(pOrigin,280.17,30.38,6.00),v60,z5,tPen\WObj:=wPaper;
    MoveL Offs(pOrigin,292.62,39.96,6.00),vTravel,z5,tPen\WObj:=wPaper;
    MoveL Offs(pOrigin,292.62,39.96,0.00),v60,z0,tPen\WObj:=wPaper;
    MoveL Offs(pOrigin,292.62,40.44,0.00),v40,z0,tPen\WObj:=wPaper;
    MoveL Offs(pOrigin,293.10,40.44,0.00),v40,z0,tPen\WObj:=wPaper;
    MoveL Offs(pOrigin,293.58,40.92,0.00),v40,z0,tPen\WObj:=wPaper;
    MoveL Offs(pOrigin,292.62,39.96,0.00),v40,z0,tPen\WObj:=wPaper;
    MoveL Offs(pOrigin,292.62,40.44,0.00),v40,z0,tPen\WObj:=wPaper;
    MoveL Offs(pOrigin,293.10,40.44,0.00),v40,z0,tPen\WObj:=wPaper;
    MoveL Offs(pOrigin,293.58,40.92,0.00),v40,z0,tPen\WObj:=wPaper;
    MoveL Offs(pOrigin,292.62,39.96,0.00),v40,fine,tPen\WObj:=wPaper;
    MoveL Offs(pOrigin,292.62,39.96,6.00),v60,z5,tPen\WObj:=wPaper;
    MoveL Offs(pOrigin,294.06,41.87,6.00),vTravel,z5,tPen\WObj:=wPaper;
    MoveL Offs(pOrigin,294.06,41.87,0.00),v60,z0,tPen\WObj:=wPaper;
    MoveL Offs(pOrigin,294.06,42.35,0.00),v40,z0,tPen\WObj:=wPaper;
    MoveL Offs(pOrigin,294.54,42.35,0.00),v40,z0,tPen\WObj:=wPaper;
    MoveL Offs(pOrigin,295.01,42.83,0.00),v40,z0,tPen\WObj:=wPaper;
    MoveL Offs(pOrigin,294.06,41.87,0.00),v40,z0,tPen\WObj:=wPaper;
    MoveL Offs(pOrigin,294.06,42.35,0.00),v40,z0,tPen\WObj:=wPaper;
    MoveL Offs(pOrigin,294.54,42.35,0.00),v40,z0,tPen\WObj:=wPaper;
    MoveL Offs(pOrigin,295.01,42.83,0.00),v40,z0,tPen\WObj:=wPaper;
    MoveL Offs(pOrigin,294.06,41.87,0.00),v40,fine,tPen\WObj:=wPaper;
    MoveL Offs(pOrigin,294.06,41.87,6.00),v60,z5,tPen\WObj:=wPaper;
    MoveL Offs(pOrigin,305.07,44.75,6.00),vTravel,z5,tPen\WObj:=wPaper;
    MoveL Offs(pOrigin,305.07,44.75,0.00),v60,z0,tPen\WObj:=wPaper;
    MoveL Offs(pOrigin,305.39,45.70,0.00),v40,z0,tPen\WObj:=wPaper;
    MoveL Offs(pOrigin,306.03,46.34,0.00),v40,z0,tPen\WObj:=wPaper;
    MoveL Offs(pOrigin,306.99,46.66,0.00),v40,z0,tPen\WObj:=wPaper;
    MoveL Offs(pOrigin,318.96,46.66,0.00),v40,z0,tPen\WObj:=wPaper;
    MoveL Offs(pOrigin,319.76,46.18,0.00),v40,z0,tPen\WObj:=wPaper;
  ENDPROC

